SPLINE
SPL {X  -133.336, Y  +773.792, Z    +0.000, E1   -47.991, E3 +231264.760}
SPL {X  -153.017, Y  +738.949, Z    +0.000, E1   -37.928, E3 +231278.164}
SPL {X  -160.146, Y  +717.846, Z    +0.000, E1   -27.412, E3 +231265.710}
SPL {X  -163.639, Y  +701.236, Z    +0.000, E1   -18.901, E3 +231271.851}
SPL {X  -165.058, Y  +689.494, Z    +0.000, E1   -11.557, E3 +231270.668}
SPL {X  -165.574, Y  +680.514, Z    +0.000, E1    -5.500, E3 +231269.912}
SPL {X  -165.650, Y  +674.881, Z    +0.000, E1    -1.215, E3 +231269.515}
SPL {X  -165.650, Y  +672.727, Z    +0.000, E1    +0.658, E3 +231268.394}
SPL {X  -165.650, Y  +669.258, Z    +0.000, E1    +5.269, E3 +231267.747}
SPL {X  -165.650, Y  +665.011, Z    +0.000, E1   +11.627, E3 +231267.634}
SPL {X  -165.650, Y  +659.446, Z    +0.000, E1   +21.123, E3 +231266.498}
SPL {X  -165.650, Y  +651.038, Z    +0.000, E1   +34.281, E3 +231266.124}
SPL {X  -165.650, Y  +635.255, Z    +0.000, E1   +53.641, E3 +231264.312}
SPL {X  -165.650, Y  +581.672, Z    +0.000, E1   +69.744, E3 +231276.720}
SPL {X  -165.650, Y  +458.048, Z    +0.000, E1   +68.782, E3 +231357.453}
ENDSPLINE

SPLINE
SPL {X  -165.650, Y  +484.472, Z    +0.000, E1   +63.918, E3 +231371.703}
ENDSPLINE

SPLINE
SPL {X  -165.650, Y  +477.868, Z    +0.000, E1   +63.324, E3 +231382.881}
SPL {X  -165.650, Y  +463.578, Z    +0.000, E1   +63.625, E3 +231395.235}
SPL {X  -165.650, Y  +453.769, Z    +0.000, E1   +63.450, E3 +231406.493}
SPL {X  -165.650, Y  +444.234, Z    +0.000, E1   +63.262, E3 +231417.666}
SPL {X  -165.650, Y  +432.479, Z    +0.000, E1   +63.557, E3 +231427.486}
SPL {X  -165.650, Y  +422.068, Z    +0.000, E1   +63.630, E3 +231437.582}
SPL {X  -165.650, Y  +411.650, Z    +0.000, E1   +63.439, E3 +231449.600}
SPL {X  -165.650, Y  +399.089, Z    +0.000, E1   +63.334, E3 +231463.325}
ENDSPLINE

SPLINE
SPL {X  -165.650, Y  +410.094, Z    +0.000, E1   +60.049, E3 +231474.043}
ENDSPLINE

SPLINE
SPL {X  -165.650, Y  +398.700, Z    +0.000, E1   +60.415, E3 +231484.941}
SPL {X  -165.650, Y  +380.643, Z    +0.000, E1   +61.187, E3 +231500.302}
SPL {X  -165.125, Y  +365.326, Z    +0.000, E1   +61.696, E3 +231513.646}
SPL {X  -164.823, Y  +361.969, Z    +0.000, E1   +60.899, E3 +231522.881}
SPL {X  -163.414, Y  +351.372, Z    +0.000, E1   +61.284, E3 +231532.143}
SPL {X  -162.189, Y  +344.818, Z    +0.000, E1   +60.900, E3 +231541.996}
SPL {X  -160.769, Y  +338.584, Z    +0.000, E1   +60.413, E3 +231552.172}
SPL {X  -157.780, Y  +328.049, Z    +0.000, E1   +60.445, E3 +231563.839}
SPL {X  -155.286, Y  +320.826, Z    +0.000, E1   +59.686, E3 +231576.395}
SPL {X  -152.445, Y  +313.689, Z    +0.000, E1   +59.490, E3 +231585.460}
SPL {X  -149.851, Y  +307.898, Z    +0.000, E1   +58.978, E3 +231594.782}
SPL {X  -146.926, Y  +301.997, Z    +0.000, E1   +58.334, E3 +231604.744}
SPL {X  -143.997, Y  +296.618, Z    +0.000, E1   +58.069, E3 +231612.002}
SPL {X  -142.530, Y  +294.089, Z    +0.000, E1   +57.567, E3 +231617.185}
SPL {X  -134.010, Y  +281.128, Z    +0.000, E1   +60.923, E3 +231615.291}
SPL {X   -93.591, Y  +241.823, Z    +0.000, E1   +55.455, E3 +231707.829}
ENDSPLINE

SPLINE
SPL {X  -110.554, Y  +255.140, Z    +0.000, E1   +52.082, E3 +231834.785}
SPL {X  -137.038, Y  +285.439, Z    +0.000, E1   +46.261, E3 +231854.524}
SPL {X  -149.954, Y  +308.117, Z    +0.000, E1   +39.560, E3 +231860.872}
SPL {X  -160.070, Y  +335.868, Z    +0.000, E1   +27.320, E3 +231855.271}
SPL {X  -163.969, Y  +354.959, Z    +0.000, E1   +17.178, E3 +231855.785}
SPL {X  -165.261, Y  +367.153, Z    +0.000, E1    +9.611, E3 +231854.937}
SPL {X  -165.600, Y  +374.440, Z    +0.000, E1    +4.699, E3 +231854.199}
SPL {X  -165.650, Y  +379.657, Z    +0.000, E1    +0.819, E3 +231853.727}
SPL {X  -165.650, Y  +381.885, Z    +0.000, E1    -1.282, E3 +231852.971}
SPL {X  -165.650, Y  +386.855, Z    +0.000, E1    -7.700, E3 +231852.390}
SPL {X  -165.650, Y  +393.198, Z    +0.000, E1   -17.733, E3 +231851.366}
SPL {X  -165.650, Y  +399.991, Z    +0.000, E1   -27.922, E3 +231852.262}
SPL {X  -165.650, Y  +411.457, Z    +0.000, E1   -45.557, E3 +231848.010}
SPL {X  -165.650, Y  +427.627, Z    +0.000, E1   -58.747, E3 +231848.644}
SPL {X  -165.650, Y  +479.770, Z    +0.000, E1   -67.621, E3 +231869.258}
SPL {X  -165.650, Y  +594.725, Z    +0.000, E1   -69.155, E3 +231936.720}
ENDSPLINE

SPLINE
SPL {X  -165.650, Y  +562.482, Z    +0.000, E1   -62.785, E3 +231956.185}
ENDSPLINE

SPLINE
SPL {X  -165.650, Y  +572.898, Z    +0.000, E1   -62.409, E3 +231970.123}
SPL {X  -165.650, Y  +586.101, Z    +0.000, E1   -62.398, E3 +231984.194}
SPL {X  -165.650, Y  +596.110, Z    +0.000, E1   -62.302, E3 +231995.635}
SPL {X  -165.650, Y  +607.052, Z    +0.000, E1   -62.387, E3 +232006.702}
SPL {X  -165.650, Y  +615.372, Z    +0.000, E1   -62.260, E3 +232016.529}
SPL {X  -165.650, Y  +628.571, Z    +0.000, E1   -62.348, E3 +232030.250}
SPL {X  -165.650, Y  +640.498, Z    +0.000, E1   -62.343, E3 +232042.871}
SPL {X  -165.650, Y  +654.166, Z    +0.000, E1   -62.507, E3 +232056.522}
SPL {X  -165.650, Y  +665.926, Z    +0.000, E1   -62.171, E3 +232071.321}
SPL {X  -165.644, Y  +676.899, Z    +0.000, E1   -62.447, E3 +232081.088}
SPL {X  -165.241, Y  +687.133, Z    +0.000, E1   -62.230, E3 +232093.791}
SPL {X  -164.056, Y  +698.425, Z    +0.000, E1   -62.113, E3 +232106.607}
SPL {X  -162.891, Y  +705.608, Z    +0.000, E1   -61.899, E3 +232115.779}
SPL {X  -160.709, Y  +715.657, Z    +0.000, E1   -61.639, E3 +232128.531}
SPL {X  -157.706, Y  +726.183, Z    +0.000, E1   -61.153, E3 +232142.914}
SPL {X  -155.057, Y  +733.785, Z    +0.000, E1   -60.834, E3 +232152.904}
SPL {X  -152.882, Y  +739.274, Z    +0.000, E1   -60.485, E3 +232160.896}
SPL {X  -149.755, Y  +746.304, Z    +0.000, E1   -59.867, E3 +232172.017}
SPL {X  -146.068, Y  +753.629, Z    +0.000, E1   -59.384, E3 +232182.377}
SPL {X  -143.119, Y  +758.908, Z    +0.000, E1   -58.828, E3 +232190.751}
SPL {X  -141.017, Y  +762.414, Z    +0.000, E1   -58.435, E3 +232196.272}
SPL {X  -134.606, Y  +772.046, Z    +0.000, E1   -61.105, E3 +232193.918}
SPL {X  -127.075, Y  +781.763, Z    +0.000, E1   -62.555, E3 +232196.233}
SPL {X   -95.057, Y  +811.161, Z    +0.000, E1   -56.196, E3 +232276.286}
SPL {X   -88.361, Y  +815.615, Z    +0.000, E1   -54.176, E3 +232322.203}
ENDSPLINE

SPLINE
SPL {X  -120.253, Y  +789.426, Z    +0.000, E1   -51.165, E3 +232429.981}
SPL {X  -143.101, Y  +758.939, Z    +0.000, E1   -44.365, E3 +232444.089}
SPL {X  -158.740, Y  +722.846, Z    +0.000, E1   -30.140, E3 +232442.127}
SPL {X  -163.639, Y  +701.236, Z    +0.000, E1   -18.901, E3 +232444.265}
SPL {X  -165.058, Y  +689.494, Z    +0.000, E1   -11.557, E3 +232443.082}
SPL {X  -165.574, Y  +680.514, Z    +0.000, E1    -5.500, E3 +232442.326}
SPL {X  -165.650, Y  +673.883, Z    +0.000, E1    -0.454, E3 +232441.337}
SPL {X  -165.650, Y  +672.004, Z    +0.000, E1    +1.620, E3 +232440.543}
SPL {X  -165.650, Y  +669.258, Z    +0.000, E1    +5.269, E3 +232440.161}
SPL {X  -165.650, Y  +665.011, Z    +0.000, E1   +11.627, E3 +232440.048}
SPL {X  -165.650, Y  +659.446, Z    +0.000, E1   +21.123, E3 +232438.912}
SPL {X  -165.650, Y  +651.038, Z    +0.000, E1   +34.281, E3 +232438.538}
SPL {X  -165.650, Y  +635.255, Z    +0.000, E1   +53.641, E3 +232436.726}
SPL {X  -165.650, Y  +581.672, Z    +0.000, E1   +69.744, E3 +232449.134}
SPL {X  -165.650, Y  +458.048, Z    +0.000, E1   +68.782, E3 +232529.866}
ENDSPLINE

SPLINE
SPL {X  -165.650, Y  +484.472, Z    +0.000, E1   +63.918, E3 +232544.117}
ENDSPLINE

SPLINE
SPL {X  -165.650, Y  +477.868, Z    +0.000, E1   +63.324, E3 +232555.295}
SPL {X  -165.650, Y  +463.578, Z    +0.000, E1   +63.625, E3 +232567.649}
SPL {X  -165.650, Y  +453.769, Z    +0.000, E1   +63.450, E3 +232578.907}
SPL {X  -165.650, Y  +444.234, Z    +0.000, E1   +63.262, E3 +232590.080}
SPL {X  -165.650, Y  +432.479, Z    +0.000, E1   +63.557, E3 +232599.900}
SPL {X  -165.650, Y  +422.068, Z    +0.000, E1   +63.630, E3 +232609.995}
SPL {X  -165.650, Y  +411.650, Z    +0.000, E1   +63.439, E3 +232622.014}
SPL {X  -165.650, Y  +399.089, Z    +0.000, E1   +63.334, E3 +232635.739}
ENDSPLINE

SPLINE
SPL {X  -165.650, Y  +410.094, Z    +0.000, E1   +60.049, E3 +232646.456}
ENDSPLINE

SPLINE
SPL {X  -165.650, Y  +398.700, Z    +0.000, E1   +60.415, E3 +232657.354}
SPL {X  -165.650, Y  +380.643, Z    +0.000, E1   +61.187, E3 +232672.716}
SPL {X  -165.125, Y  +365.326, Z    +0.000, E1   +61.696, E3 +232686.060}
SPL {X  -164.823, Y  +361.969, Z    +0.000, E1   +60.899, E3 +232695.294}
SPL {X  -163.414, Y  +351.372, Z    +0.000, E1   +61.284, E3 +232704.557}
SPL {X  -162.189, Y  +344.818, Z    +0.000, E1   +60.900, E3 +232714.410}
SPL {X  -160.769, Y  +338.584, Z    +0.000, E1   +60.413, E3 +232724.586}
SPL {X  -157.780, Y  +328.049, Z    +0.000, E1   +60.445, E3 +232736.253}
SPL {X  -155.286, Y  +320.826, Z    +0.000, E1   +59.686, E3 +232748.809}
SPL {X  -152.445, Y  +313.689, Z    +0.000, E1   +59.490, E3 +232757.874}
SPL {X  -150.678, Y  +309.680, Z    +0.000, E1   +58.971, E3 +232765.186}
SPL {X  -148.010, Y  +304.117, Z    +0.000, E1   +58.696, E3 +232772.933}
SPL {X  -144.822, Y  +298.086, Z    +0.000, E1   +58.093, E3 +232782.715}
SPL {X  -142.530, Y  +294.089, Z    +0.000, E1   +57.567, E3 +232789.599}
SPL {X  -136.453, Y  +284.583, Z    +0.000, E1   +60.257, E3 +232787.410}
SPL {X  -128.205, Y  +273.602, Z    +0.000, E1   +62.388, E3 +232788.113}
SPL {X   -93.591, Y  +241.823, Z    +0.000, E1   +55.455, E3 +232880.243}
ENDSPLINE

SPLINE
SPL {X  -110.554, Y  +255.140, Z    +0.000, E1   +52.082, E3 +233007.199}
SPL {X  -137.038, Y  +285.439, Z    +0.000, E1   +46.261, E3 +233026.938}
SPL {X  -149.954, Y  +308.117, Z    +0.000, E1   +39.560, E3 +233033.286}
SPL {X  -160.070, Y  +335.868, Z    +0.000, E1   +27.320, E3 +233027.685}
SPL {X  -163.969, Y  +354.959, Z    +0.000, E1   +17.178, E3 +233028.199}
SPL {X  -165.261, Y  +367.153, Z    +0.000, E1    +9.611, E3 +233027.351}
SPL {X  -165.600, Y  +374.440, Z    +0.000, E1    +4.699, E3 +233026.612}
SPL {X  -165.650, Y  +379.657, Z    +0.000, E1    +0.819, E3 +233026.141}
SPL {X  -165.650, Y  +381.885, Z    +0.000, E1    -1.282, E3 +233025.385}
SPL {X  -165.650, Y  +386.855, Z    +0.000, E1    -7.700, E3 +233024.804}
SPL {X  -165.650, Y  +393.198, Z    +0.000, E1   -17.733, E3 +233023.780}
SPL {X  -165.650, Y  +399.991, Z    +0.000, E1   -27.922, E3 +233024.676}
SPL {X  -165.650, Y  +411.457, Z    +0.000, E1   -45.557, E3 +233020.424}
SPL {X  -165.650, Y  +427.627, Z    +0.000, E1   -58.747, E3 +233021.058}
SPL {X  -165.650, Y  +479.770, Z    +0.000, E1   -67.621, E3 +233041.672}
SPL {X  -165.650, Y  +594.725, Z    +0.000, E1   -69.155, E3 +233109.134}
ENDSPLINE

SPLINE
SPL {X  -165.650, Y  +565.175, Z    +0.000, E1   -62.653, E3 +233132.624}
ENDSPLINE

SPLINE
SPL {X  -165.650, Y  +576.067, Z    +0.000, E1   -62.373, E3 +233146.025}
SPL {X  -165.650, Y  +586.101, Z    +0.000, E1   -62.398, E3 +233156.608}
SPL {X  -165.650, Y  +596.110, Z    +0.000, E1   -62.302, E3 +233168.048}
SPL {X  -165.650, Y  +607.052, Z    +0.000, E1   -62.387, E3 +233179.116}
SPL {X  -165.650, Y  +618.920, Z    +0.000, E1   -62.340, E3 +233192.306}
SPL {X  -165.650, Y  +635.445, Z    +0.000, E1   -62.341, E3 +233210.106}
SPL {X  -165.650, Y  +654.166, Z    +0.000, E1   -62.507, E3 +233228.936}
SPL {X  -165.650, Y  +665.926, Z    +0.000, E1   -62.171, E3 +233243.734}
SPL {X  -165.644, Y  +676.899, Z    +0.000, E1   -62.447, E3 +233253.502}
SPL {X  -165.241, Y  +687.133, Z    +0.000, E1   -62.230, E3 +233266.204}
SPL {X  -164.056, Y  +698.425, Z    +0.000, E1   -62.113, E3 +233279.021}
SPL {X  -162.891, Y  +705.608, Z    +0.000, E1   -61.899, E3 +233288.193}
SPL {X  -161.308, Y  +713.180, Z    +0.000, E1   -61.813, E3 +233296.887}
SPL {X  -159.339, Y  +720.787, Z    +0.000, E1   -61.452, E3 +233307.582}
SPL {X  -156.103, Y  +730.922, Z    +0.000, E1   -60.875, E3 +233322.128}
SPL {X  -152.882, Y  +739.274, Z    +0.000, E1   -60.485, E3 +233333.310}
SPL {X  -150.387, Y  +744.953, Z    +0.000, E1   -60.023, E3 +233341.985}
SPL {X  -147.728, Y  +750.443, Z    +0.000, E1   -59.568, E3 +233350.369}
SPL {X  -143.895, Y  +757.561, Z    +0.000, E1   -58.980, E3 +233361.105}
SPL {X  -141.017, Y  +762.414, Z    +0.000, E1   -58.435, E3 +233368.685}
SPL {X  -132.386, Y  +775.068, Z    +0.000, E1   -61.559, E3 +233367.071}
SPL {X   -89.692, Y  +814.767, Z    +0.000, E1   -54.641, E3 +233481.120}
ENDSPLINE

SPLINE
SPL {X  -133.336, Y  +773.792, Z    +0.000, E1   -47.991, E3 +233609.587}
SPL {X  -153.017, Y  +738.949, Z    +0.000, E1   -37.928, E3 +233622.991}
SPL {X  -160.146, Y  +717.846, Z    +0.000, E1   -27.412, E3 +233610.537}
SPL {X  -163.639, Y  +701.236, Z    +0.000, E1   -18.901, E3 +233616.679}
SPL {X  -165.058, Y  +689.494, Z    +0.000, E1   -11.557, E3 +233615.496}
SPL {X  -165.574, Y  +680.514, Z    +0.000, E1    -5.500, E3 +233614.739}
SPL {X  -165.650, Y  +674.881, Z    +0.000, E1    -1.215, E3 +233614.342}
SPL {X  -165.650, Y  +673.425, Z    +0.000, E1    +0.051, E3 +233613.478}
SPL {X  -165.650, Y  +672.004, Z    +0.000, E1    +1.620, E3 +233612.956}
SPL {X  -165.650, Y  +669.258, Z    +0.000, E1    +5.269, E3 +233612.575}
SPL {X  -165.650, Y  +665.011, Z    +0.000, E1   +11.627, E3 +233612.462}
SPL {X  -165.650, Y  +659.446, Z    +0.000, E1   +21.123, E3 +233611.326}
SPL {X  -165.650, Y  +654.020, Z    +0.000, E1   +29.754, E3 +233611.481}
SPL {X  -165.650, Y  +644.843, Z    +0.000, E1   +43.427, E3 +233609.807}
SPL {X  -165.650, Y  +632.102, Z    +0.000, E1   +56.225, E3 +233609.155}
SPL {X  -165.650, Y  +581.672, Z    +0.000, E1   +69.744, E3 +233621.547}
SPL {X  -165.650, Y  +458.048, Z    +0.000, E1   +68.782, E3 +233702.280}
ENDSPLINE

SPLINE
SPL {X  -165.650, Y  +484.472, Z    +0.000, E1   +63.918, E3 +233716.531}
ENDSPLINE

SPLINE
SPL {X  -165.650, Y  +477.868, Z    +0.000, E1   +63.324, E3 +233727.708}
SPL {X  -165.650, Y  +463.578, Z    +0.000, E1   +63.625, E3 +233740.062}
SPL {X  -165.650, Y  +453.769, Z    +0.000, E1   +63.450, E3 +233751.321}
SPL {X  -165.650, Y  +444.234, Z    +0.000, E1   +63.262, E3 +233762.494}
SPL {X  -165.650, Y  +432.479, Z    +0.000, E1   +63.557, E3 +233772.314}
SPL {X  -165.650, Y  +422.068, Z    +0.000, E1   +63.630, E3 +233782.409}
SPL {X  -165.650, Y  +409.231, Z    +0.000, E1   +63.364, E3 +233797.658}
SPL {X  -165.650, Y  +395.008, Z    +0.000, E1   +63.445, E3 +233811.421}
ENDSPLINE

SPLINE
SPL {X  -165.650, Y  +410.094, Z    +0.000, E1   +60.049, E3 +233818.870}
ENDSPLINE

SPLINE
SPL {X  -165.650, Y  +398.700, Z    +0.000, E1   +60.415, E3 +233829.768}
SPL {X  -165.650, Y  +382.616, Z    +0.000, E1   +61.427, E3 +233840.987}
SPL {X  -165.650, Y  +379.013, Z    +0.000, E1   +60.888, E3 +233848.809}
SPL {X  -165.125, Y  +365.326, Z    +0.000, E1   +61.696, E3 +233858.473}
SPL {X  -164.823, Y  +361.969, Z    +0.000, E1   +60.899, E3 +233867.708}
SPL {X  -163.414, Y  +351.372, Z    +0.000, E1   +61.284, E3 +233876.971}
SPL {X  -162.189, Y  +344.818, Z    +0.000, E1   +60.900, E3 +233886.824}
SPL {X  -160.769, Y  +338.584, Z    +0.000, E1   +60.413, E3 +233897.000}
SPL {X  -157.780, Y  +328.049, Z    +0.000, E1   +60.445, E3 +233908.667}
SPL {X  -155.286, Y  +320.826, Z    +0.000, E1   +59.686, E3 +233921.222}
SPL {X  -152.445, Y  +313.689, Z    +0.000, E1   +59.490, E3 +233930.288}
SPL {X  -149.851, Y  +307.898, Z    +0.000, E1   +58.978, E3 +233939.610}
SPL {X  -146.926, Y  +301.997, Z    +0.000, E1   +58.334, E3 +233949.571}
SPL {X  -143.281, Y  +295.370, Z    +0.000, E1   +57.860, E3 +233959.340}
SPL {X  -136.453, Y  +284.583, Z    +0.000, E1   +60.257, E3 +233959.824}
SPL {X  -128.205, Y  +273.602, Z    +0.000, E1   +62.388, E3 +233960.527}
SPL {X   -93.591, Y  +241.823, Z    +0.000, E1   +55.455, E3 +234052.656}
ENDSPLINE

SPLINE
SPL {X  -110.554, Y  +255.140, Z    +0.000, E1   +52.082, E3 +234179.612}
SPL {X  -137.038, Y  +285.439, Z    +0.000, E1   +46.261, E3 +234199.352}
SPL {X  -149.954, Y  +308.117, Z    +0.000, E1   +39.560, E3 +234205.700}
SPL {X  -160.070, Y  +335.868, Z    +0.000, E1   +27.320, E3 +234200.098}
SPL {X  -163.969, Y  +354.959, Z    +0.000, E1   +17.178, E3 +234200.613}
SPL {X  -165.261, Y  +367.153, Z    +0.000, E1    +9.611, E3 +234199.765}
SPL {X  -165.600, Y  +374.440, Z    +0.000, E1    +4.699, E3 +234199.026}
SPL {X  -165.650, Y  +379.657, Z    +0.000, E1    +0.819, E3 +234198.555}
SPL {X  -165.650, Y  +381.885, Z    +0.000, E1    -1.282, E3 +234197.799}
SPL {X  -165.650, Y  +385.555, Z    +0.000, E1    -6.051, E3 +234196.944}
SPL {X  -165.650, Y  +388.884, Z    +0.000, E1   -10.835, E3 +234197.644}
SPL {X  -165.650, Y  +393.198, Z    +0.000, E1   -17.733, E3 +234196.194}
SPL {X  -165.650, Y  +399.991, Z    +0.000, E1   -27.922, E3 +234197.090}
SPL {X  -165.650, Y  +409.148, Z    +0.000, E1   -43.235, E3 +234192.476}
SPL {X  -165.650, Y  +420.563, Z    +0.000, E1   -54.059, E3 +234193.034}
SPL {X  -165.650, Y  +436.566, Z    +0.000, E1   -62.888, E3 +234194.747}
SPL {X  -165.650, Y  +479.770, Z    +0.000, E1   -67.621, E3 +234214.085}
SPL {X  -165.650, Y  +594.725, Z    +0.000, E1   -69.155, E3 +234281.547}
ENDSPLINE

SPLINE
SPL {X  -165.650, Y  +565.175, Z    +0.000, E1   -62.653, E3 +234305.038}
ENDSPLINE

SPLINE
SPL {X  -165.650, Y  +576.067, Z    +0.000, E1   -62.373, E3 +234318.439}
SPL {X  -165.650, Y  +586.101, Z    +0.000, E1   -62.398, E3 +234329.021}
SPL {X  -165.650, Y  +596.110, Z    +0.000, E1   -62.302, E3 +234340.462}
SPL {X  -165.650, Y  +607.052, Z    +0.000, E1   -62.387, E3 +234351.529}
SPL {X  -165.650, Y  +618.920, Z    +0.000, E1   -62.340, E3 +234364.720}
SPL {X  -165.650, Y  +635.445, Z    +0.000, E1   -62.341, E3 +234382.520}
SPL {X  -165.650, Y  +654.166, Z    +0.000, E1   -62.507, E3 +234401.350}
SPL {X  -165.650, Y  +665.926, Z    +0.000, E1   -62.171, E3 +234416.148}
SPL {X  -165.600, Y  +679.566, Z    +0.000, E1   -62.408, E3 +234429.186}
SPL {X  -165.066, Y  +689.394, Z    +0.000, E1   -62.143, E3 +234441.515}
SPL {X  -164.056, Y  +698.425, Z    +0.000, E1   -62.113, E3 +234451.435}
SPL {X  -162.891, Y  +705.608, Z    +0.000, E1   -61.899, E3 +234460.607}
SPL {X  -161.308, Y  +713.180, Z    +0.000, E1   -61.813, E3 +234469.300}
SPL {X  -159.339, Y  +720.787, Z    +0.000, E1   -61.452, E3 +234479.995}
SPL {X  -156.103, Y  +730.922, Z    +0.000, E1   -60.875, E3 +234494.542}
SPL {X  -152.882, Y  +739.274, Z    +0.000, E1   -60.485, E3 +234505.724}
SPL {X  -150.387, Y  +744.953, Z    +0.000, E1   -60.023, E3 +234514.399}
SPL {X  -147.728, Y  +750.443, Z    +0.000, E1   -59.568, E3 +234522.783}
SPL {X  -143.895, Y  +757.561, Z    +0.000, E1   -58.980, E3 +234533.519}
SPL {X  -141.017, Y  +762.414, Z    +0.000, E1   -58.435, E3 +234541.099}
SPL {X  -132.386, Y  +775.068, Z    +0.000, E1   -61.559, E3 +234539.485}
SPL {X   -89.692, Y  +814.767, Z    +0.000, E1   -54.641, E3 +234653.534}
ENDSPLINE

SPLINE
SPL {X  -133.336, Y  +773.792, Z    +0.000, E1   -47.991, E3 +234782.001}
SPL {X  -153.017, Y  +738.949, Z    +0.000, E1   -37.928, E3 +234795.405}
SPL {X  -160.146, Y  +717.846, Z    +0.000, E1   -27.412, E3 +234782.951}
SPL {X  -163.639, Y  +701.236, Z    +0.000, E1   -18.901, E3 +234789.093}
SPL {X  -165.058, Y  +689.494, Z    +0.000, E1   -11.557, E3 +234787.910}
SPL {X  -165.574, Y  +680.514, Z    +0.000, E1    -5.500, E3 +234787.153}
SPL {X  -165.650, Y  +673.883, Z    +0.000, E1    -0.454, E3 +234786.164}
SPL {X  -165.650, Y  +672.004, Z    +0.000, E1    +1.620, E3 +234785.370}
SPL {X  -165.650, Y  +669.258, Z    +0.000, E1    +5.269, E3 +234784.988}
SPL {X  -165.650, Y  +665.011, Z    +0.000, E1   +11.627, E3 +234784.876}
SPL {X  -165.650, Y  +659.446, Z    +0.000, E1   +21.123, E3 +234783.740}
SPL {X  -165.650, Y  +654.020, Z    +0.000, E1   +29.754, E3 +234783.894}
SPL {X  -165.650, Y  +644.843, Z    +0.000, E1   +43.427, E3 +234782.220}
SPL {X  -165.650, Y  +632.102, Z    +0.000, E1   +56.225, E3 +234781.569}
SPL {X  -165.650, Y  +581.672, Z    +0.000, E1   +69.744, E3 +234793.961}
SPL {X  -165.650, Y  +458.048, Z    +0.000, E1   +68.782, E3 +234874.694}
ENDSPLINE

SPLINE
SPL {X  -165.650, Y  +484.472, Z    +0.000, E1   +63.918, E3 +234888.945}
ENDSPLINE

SPLINE
SPL {X  -165.650, Y  +477.868, Z    +0.000, E1   +63.324, E3 +234900.122}
SPL {X  -165.650, Y  +463.578, Z    +0.000, E1   +63.625, E3 +234912.476}
SPL {X  -165.650, Y  +453.769, Z    +0.000, E1   +63.450, E3 +234923.735}
SPL {X  -165.650, Y  +444.234, Z    +0.000, E1   +63.262, E3 +234934.908}
SPL {X  -165.650, Y  +432.479, Z    +0.000, E1   +63.557, E3 +234944.728}
SPL {X  -165.650, Y  +422.068, Z    +0.000, E1   +63.630, E3 +234954.823}
SPL {X  -165.650, Y  +409.231, Z    +0.000, E1   +63.364, E3 +234970.071}
SPL {X  -165.650, Y  +395.008, Z    +0.000, E1   +63.445, E3 +234983.835}
ENDSPLINE

SPLINE
SPL {X  -165.650, Y  +410.094, Z    +0.000, E1   +60.049, E3 +234991.284}
ENDSPLINE

SPLINE
SPL {X  -165.650, Y  +398.700, Z    +0.000, E1   +60.415, E3 +235002.182}
SPL {X  -165.650, Y  +382.616, Z    +0.000, E1   +61.427, E3 +235013.400}
SPL {X  -165.650, Y  +379.013, Z    +0.000, E1   +60.888, E3 +235021.223}
SPL {X  -165.125, Y  +365.326, Z    +0.000, E1   +61.696, E3 +235030.887}
SPL {X  -164.823, Y  +361.969, Z    +0.000, E1   +60.899, E3 +235040.122}
SPL {X  -163.414, Y  +351.372, Z    +0.000, E1   +61.284, E3 +235049.385}
SPL {X  -162.189, Y  +344.818, Z    +0.000, E1   +60.900, E3 +235059.238}
SPL {X  -160.769, Y  +338.584, Z    +0.000, E1   +60.413, E3 +235069.414}
SPL {X  -157.780, Y  +328.049, Z    +0.000, E1   +60.445, E3 +235081.081}
SPL {X  -155.286, Y  +320.826, Z    +0.000, E1   +59.686, E3 +235093.636}
SPL {X  -152.445, Y  +313.689, Z    +0.000, E1   +59.490, E3 +235102.702}
SPL {X  -149.851, Y  +307.898, Z    +0.000, E1   +58.978, E3 +235112.024}
SPL {X  -146.926, Y  +301.997, Z    +0.000, E1   +58.334, E3 +235121.985}
SPL {X  -143.997, Y  +296.618, Z    +0.000, E1   +58.069, E3 +235129.243}
SPL {X  -142.530, Y  +294.089, Z    +0.000, E1   +57.567, E3 +235134.426}
SPL {X  -134.010, Y  +281.128, Z    +0.000, E1   +60.923, E3 +235132.532}
SPL {X   -93.591, Y  +241.823, Z    +0.000, E1   +55.455, E3 +235225.070}
ENDSPLINE

SPLINE
SPL {X  -110.554, Y  +255.140, Z    +0.000, E1   +52.082, E3 +235352.026}
SPL {X  -144.988, Y  +298.385, Z    +0.000, E1   +42.755, E3 +235375.845}
SPL {X  -160.070, Y  +335.868, Z    +0.000, E1   +27.320, E3 +235372.512}
SPL {X  -163.969, Y  +354.959, Z    +0.000, E1   +17.178, E3 +235373.026}
SPL {X  -165.261, Y  +367.153, Z    +0.000, E1    +9.611, E3 +235372.179}
SPL {X  -165.600, Y  +374.440, Z    +0.000, E1    +4.699, E3 +235371.440}
SPL {X  -165.650, Y  +379.657, Z    +0.000, E1    +0.819, E3 +235370.968}
SPL {X  -165.650, Y  +381.885, Z    +0.000, E1    -1.282, E3 +235370.213}
SPL {X  -165.650, Y  +386.855, Z    +0.000, E1    -7.700, E3 +235369.632}
SPL {X  -165.650, Y  +393.198, Z    +0.000, E1   -17.733, E3 +235368.608}
SPL {X  -165.650, Y  +399.991, Z    +0.000, E1   -27.922, E3 +235369.503}
SPL {X  -165.650, Y  +409.148, Z    +0.000, E1   -43.235, E3 +235364.890}
SPL {X  -165.650, Y  +420.563, Z    +0.000, E1   -54.059, E3 +235365.447}
SPL {X  -165.650, Y  +436.566, Z    +0.000, E1   -62.888, E3 +235367.160}
SPL {X  -165.650, Y  +479.770, Z    +0.000, E1   -67.621, E3 +235386.499}
SPL {X  -165.650, Y  +594.725, Z    +0.000, E1   -69.155, E3 +235453.961}
ENDSPLINE

SPLINE
SPL {X  -165.650, Y  +565.175, Z    +0.000, E1   -62.653, E3 +235477.452}
ENDSPLINE

SPLINE
SPL {X  -165.650, Y  +576.067, Z    +0.000, E1   -62.373, E3 +235490.853}
SPL {X  -165.650, Y  +586.101, Z    +0.000, E1   -62.398, E3 +235501.435}
SPL {X  -165.650, Y  +596.110, Z    +0.000, E1   -62.302, E3 +235512.876}
SPL {X  -165.650, Y  +607.052, Z    +0.000, E1   -62.387, E3 +235523.943}
SPL {X  -165.650, Y  +618.920, Z    +0.000, E1   -62.340, E3 +235537.133}
SPL {X  -165.650, Y  +635.445, Z    +0.000, E1   -62.341, E3 +235554.934}
SPL {X  -165.650, Y  +654.166, Z    +0.000, E1   -62.507, E3 +235573.764}
SPL {X  -165.650, Y  +665.926, Z    +0.000, E1   -62.171, E3 +235588.562}
SPL {X  -165.644, Y  +676.899, Z    +0.000, E1   -62.447, E3 +235598.329}
SPL {X  -165.241, Y  +687.133, Z    +0.000, E1   -62.230, E3 +235611.032}
SPL {X  -164.056, Y  +698.425, Z    +0.000, E1   -62.113, E3 +235623.849}
SPL {X  -162.891, Y  +705.608, Z    +0.000, E1   -61.899, E3 +235633.020}
SPL {X  -160.709, Y  +715.657, Z    +0.000, E1   -61.639, E3 +235645.772}
SPL {X  -157.706, Y  +726.183, Z    +0.000, E1   -61.153, E3 +235660.155}
SPL {X  -155.057, Y  +733.785, Z    +0.000, E1   -60.834, E3 +235670.145}
SPL {X  -152.882, Y  +739.274, Z    +0.000, E1   -60.485, E3 +235678.137}
SPL {X  -150.387, Y  +744.953, Z    +0.000, E1   -60.023, E3 +235686.812}
SPL {X  -147.728, Y  +750.443, Z    +0.000, E1   -59.568, E3 +235695.196}
SPL {X  -143.895, Y  +757.561, Z    +0.000, E1   -58.980, E3 +235705.933}
SPL {X  -141.017, Y  +762.414, Z    +0.000, E1   -58.435, E3 +235713.513}
SPL {X  -134.606, Y  +772.046, Z    +0.000, E1   -61.105, E3 +235711.160}
SPL {X  -127.075, Y  +781.763, Z    +0.000, E1   -62.555, E3 +235713.474}
SPL {X   -89.692, Y  +814.767, Z    +0.000, E1   -54.641, E3 +235825.948}
ENDSPLINE

SPLINE
SPL {X  -133.336, Y  +773.792, Z    +0.000, E1   -47.991, E3 +235954.415}
SPL {X  -153.017, Y  +738.949, Z    +0.000, E1   -37.928, E3 +235967.819}
SPL {X  -160.146, Y  +717.846, Z    +0.000, E1   -27.412, E3 +235955.365}
SPL {X  -163.639, Y  +701.236, Z    +0.000, E1   -18.901, E3 +235961.506}
SPL {X  -165.380, Y  +684.951, Z    +0.000, E1    -8.606, E3 +235959.764}
SPL {X  -165.650, Y  +675.640, Z    +0.000, E1    -1.874, E3 +235959.300}
SPL {X  -165.650, Y  +672.727, Z    +0.000, E1    +0.658, E3 +235958.049}
SPL {X  -165.650, Y  +669.258, Z    +0.000, E1    +5.269, E3 +235957.402}
SPL {X  -165.650, Y  +665.011, Z    +0.000, E1   +11.627, E3 +235957.289}
SPL {X  -165.650, Y  +659.446, Z    +0.000, E1   +21.123, E3 +235956.154}
SPL {X  -165.650, Y  +654.020, Z    +0.000, E1   +29.754, E3 +235956.308}
SPL {X  -165.650, Y  +644.843, Z    +0.000, E1   +43.427, E3 +235954.634}
SPL {X  -165.650, Y  +632.102, Z    +0.000, E1   +56.225, E3 +235953.983}
SPL {X  -165.650, Y  +581.672, Z    +0.000, E1   +69.744, E3 +235966.375}
SPL {X  -165.650, Y  +455.882, Z    +0.000, E1   +70.075, E3 +236038.640}
ENDSPLINE

SPLINE
SPL {X  -165.650, Y  +480.501, Z    +0.000, E1   +64.561, E3 +236060.609}
ENDSPLINE

SPLINE
SPL {X  -165.650, Y  +477.868, Z    +0.000, E1   +63.324, E3 +236072.536}
SPL {X  -165.650, Y  +463.578, Z    +0.000, E1   +63.625, E3 +236084.890}
SPL {X  -165.650, Y  +453.769, Z    +0.000, E1   +63.450, E3 +236096.149}
SPL {X  -165.650, Y  +444.234, Z    +0.000, E1   +63.262, E3 +236107.321}
SPL {X  -165.650, Y  +432.479, Z    +0.000, E1   +63.557, E3 +236117.141}
SPL {X  -165.650, Y  +422.068, Z    +0.000, E1   +63.630, E3 +236127.237}
SPL {X  -165.650, Y  +409.231, Z    +0.000, E1   +63.364, E3 +236142.485}
SPL {X  -165.650, Y  +395.008, Z    +0.000, E1   +63.445, E3 +236156.249}
ENDSPLINE

SPLINE
SPL {X  -165.650, Y  +410.094, Z    +0.000, E1   +60.049, E3 +236163.698}
ENDSPLINE

SPLINE
SPL {X  -165.650, Y  +398.700, Z    +0.000, E1   +60.415, E3 +236174.596}
SPL {X  -165.650, Y  +380.643, Z    +0.000, E1   +61.187, E3 +236189.957}
SPL {X  -165.125, Y  +365.326, Z    +0.000, E1   +61.696, E3 +236203.301}
SPL {X  -164.823, Y  +361.969, Z    +0.000, E1   +60.899, E3 +236212.536}
SPL {X  -163.414, Y  +351.372, Z    +0.000, E1   +61.284, E3 +236221.798}
SPL {X  -162.189, Y  +344.818, Z    +0.000, E1   +60.900, E3 +236231.652}
SPL {X  -160.769, Y  +338.584, Z    +0.000, E1   +60.413, E3 +236241.828}
SPL {X  -157.780, Y  +328.049, Z    +0.000, E1   +60.445, E3 +236253.494}
SPL {X  -155.286, Y  +320.826, Z    +0.000, E1   +59.686, E3 +236266.050}
SPL {X  -152.445, Y  +313.689, Z    +0.000, E1   +59.490, E3 +236275.115}
SPL {X  -149.851, Y  +307.898, Z    +0.000, E1   +58.978, E3 +236284.438}
SPL {X  -146.926, Y  +301.997, Z    +0.000, E1   +58.334, E3 +236294.399}
SPL {X  -143.281, Y  +295.370, Z    +0.000, E1   +57.860, E3 +236304.167}
SPL {X  -134.010, Y  +281.128, Z    +0.000, E1   +60.923, E3 +236304.946}
SPL {X   -93.591, Y  +241.823, Z    +0.000, E1   +55.455, E3 +236397.484}
ENDSPLINE

SPLINE
SPL {X  -110.554, Y  +255.140, Z    +0.000, E1   +52.082, E3 +236524.440}
SPL {X  -137.038, Y  +285.439, Z    +0.000, E1   +46.261, E3 +236544.180}
SPL {X  -149.954, Y  +308.117, Z    +0.000, E1   +39.560, E3 +236550.527}
SPL {X  -160.070, Y  +335.868, Z    +0.000, E1   +27.320, E3 +236544.926}
SPL {X  -163.969, Y  +354.959, Z    +0.000, E1   +17.178, E3 +236545.440}
SPL {X  -165.261, Y  +367.153, Z    +0.000, E1    +9.611, E3 +236544.593}
SPL {X  -165.600, Y  +374.440, Z    +0.000, E1    +4.699, E3 +236543.854}
SPL {X  -165.650, Y  +379.657, Z    +0.000, E1    +0.819, E3 +236543.382}
SPL {X  -165.650, Y  +381.885, Z    +0.000, E1    -1.282, E3 +236542.626}
SPL {X  -165.650, Y  +386.855, Z    +0.000, E1    -7.700, E3 +236542.045}
SPL {X  -165.650, Y  +393.198, Z    +0.000, E1   -17.733, E3 +236541.021}
SPL {X  -165.650, Y  +399.991, Z    +0.000, E1   -27.922, E3 +236541.917}
SPL {X  -165.650, Y  +409.148, Z    +0.000, E1   -43.235, E3 +236537.303}
SPL {X  -165.650, Y  +420.563, Z    +0.000, E1   -54.059, E3 +236537.861}
SPL {X  -165.650, Y  +436.566, Z    +0.000, E1   -62.888, E3 +236539.574}
SPL {X  -165.650, Y  +479.770, Z    +0.000, E1   -67.621, E3 +236558.913}
SPL {X  -165.650, Y  +594.725, Z    +0.000, E1   -69.155, E3 +236626.375}
ENDSPLINE

SPLINE
SPL {X  -165.650, Y  +565.175, Z    +0.000, E1   -62.653, E3 +236649.866}
ENDSPLINE

SPLINE
SPL {X  -165.650, Y  +576.067, Z    +0.000, E1   -62.373, E3 +236663.267}
SPL {X  -165.650, Y  +586.101, Z    +0.000, E1   -62.398, E3 +236673.849}
SPL {X  -165.650, Y  +596.110, Z    +0.000, E1   -62.302, E3 +236685.290}
SPL {X  -165.650, Y  +607.052, Z    +0.000, E1   -62.387, E3 +236696.357}
SPL {X  -165.650, Y  +618.920, Z    +0.000, E1   -62.340, E3 +236709.547}
SPL {X  -165.650, Y  +631.247, Z    +0.000, E1   -62.270, E3 +236723.164}
SPL {X  -165.650, Y  +645.288, Z    +0.000, E1   -62.475, E3 +236736.844}
SPL {X  -165.650, Y  +657.265, Z    +0.000, E1   -62.410, E3 +236749.962}
SPL {X  -165.650, Y  +665.926, Z    +0.000, E1   -62.171, E3 +236760.976}
SPL {X  -165.644, Y  +676.899, Z    +0.000, E1   -62.447, E3 +236770.743}
SPL {X  -165.241, Y  +687.133, Z    +0.000, E1   -62.230, E3 +236783.446}
SPL {X  -164.056, Y  +698.425, Z    +0.000, E1   -62.113, E3 +236796.263}
SPL {X  -162.891, Y  +705.608, Z    +0.000, E1   -61.899, E3 +236805.434}
SPL {X  -160.709, Y  +715.657, Z    +0.000, E1   -61.639, E3 +236818.186}
SPL {X  -157.706, Y  +726.183, Z    +0.000, E1   -61.153, E3 +236832.569}
SPL {X  -155.057, Y  +733.785, Z    +0.000, E1   -60.834, E3 +236842.559}
SPL {X  -152.882, Y  +739.274, Z    +0.000, E1   -60.485, E3 +236850.551}
SPL {X  -150.387, Y  +744.953, Z    +0.000, E1   -60.023, E3 +236859.226}
SPL {X  -146.839, Y  +752.170, Z    +0.000, E1   -59.458, E3 +236870.185}
SPL {X  -142.415, Y  +760.104, Z    +0.000, E1   -58.730, E3 +236882.244}
SPL {X  -132.386, Y  +775.068, Z    +0.000, E1   -61.559, E3 +236884.312}
SPL {X   -89.692, Y  +814.767, Z    +0.000, E1   -54.641, E3 +236998.362}
ENDSPLINE

SPLINE
SPL {X  -120.253, Y  +789.426, Z    +0.000, E1   -51.165, E3 +237119.636}
SPL {X  -143.101, Y  +758.939, Z    +0.000, E1   -44.365, E3 +237133.744}
SPL {X  -158.740, Y  +722.846, Z    +0.000, E1   -30.140, E3 +237131.782}
SPL {X  -163.639, Y  +701.236, Z    +0.000, E1   -18.901, E3 +237133.920}
SPL {X  -165.058, Y  +689.494, Z    +0.000, E1   -11.557, E3 +237132.737}
SPL {X  -165.574, Y  +680.514, Z    +0.000, E1    -5.500, E3 +237131.981}
SPL {X  -165.650, Y  +673.883, Z    +0.000, E1    -0.454, E3 +237130.992}
SPL {X  -165.650, Y  +672.004, Z    +0.000, E1    +1.620, E3 +237130.198}
SPL {X  -165.650, Y  +669.258, Z    +0.000, E1    +5.269, E3 +237129.816}
SPL {X  -165.650, Y  +665.011, Z    +0.000, E1   +11.627, E3 +237129.703}
SPL {X  -165.650, Y  +659.446, Z    +0.000, E1   +21.123, E3 +237128.567}
SPL {X  -165.650, Y  +654.020, Z    +0.000, E1   +29.754, E3 +237128.722}
SPL {X  -165.650, Y  +644.843, Z    +0.000, E1   +43.427, E3 +237127.048}
SPL {X  -165.650, Y  +632.102, Z    +0.000, E1   +56.225, E3 +237126.397}
SPL {X  -165.650, Y  +581.672, Z    +0.000, E1   +69.744, E3 +237138.789}
SPL {X  -165.650, Y  +458.048, Z    +0.000, E1   +68.782, E3 +237219.522}
ENDSPLINE

SPLINE
SPL {X  -165.650, Y  +484.472, Z    +0.000, E1   +63.918, E3 +237233.772}
ENDSPLINE

SPLINE
SPL {X  -165.650, Y  +477.868, Z    +0.000, E1   +63.324, E3 +237244.950}
SPL {X  -165.650, Y  +463.578, Z    +0.000, E1   +63.625, E3 +237257.304}
SPL {X  -165.650, Y  +453.769, Z    +0.000, E1   +63.450, E3 +237268.562}
SPL {X  -165.650, Y  +444.234, Z    +0.000, E1   +63.262, E3 +237279.735}
SPL {X  -165.650, Y  +432.479, Z    +0.000, E1   +63.557, E3 +237289.555}
SPL {X  -165.650, Y  +422.068, Z    +0.000, E1   +63.630, E3 +237299.650}
SPL {X  -165.650, Y  +411.650, Z    +0.000, E1   +63.439, E3 +237311.669}
SPL {X  -165.650, Y  +399.089, Z    +0.000, E1   +63.334, E3 +237325.394}
ENDSPLINE

SPLINE
SPL {X  -165.650, Y  +410.094, Z    +0.000, E1   +60.049, E3 +237336.112}
ENDSPLINE

SPLINE
SPL {X  -165.650, Y  +398.700, Z    +0.000, E1   +60.415, E3 +237347.010}
SPL {X  -165.650, Y  +380.643, Z    +0.000, E1   +61.187, E3 +237362.371}
SPL {X  -165.125, Y  +365.326, Z    +0.000, E1   +61.696, E3 +237375.715}
SPL {X  -164.823, Y  +361.969, Z    +0.000, E1   +60.899, E3 +237384.950}
SPL {X  -163.414, Y  +351.372, Z    +0.000, E1   +61.284, E3 +237394.212}
SPL {X  -162.189, Y  +344.818, Z    +0.000, E1   +60.900, E3 +237404.065}
SPL {X  -160.769, Y  +338.584, Z    +0.000, E1   +60.413, E3 +237414.241}
SPL {X  -157.780, Y  +328.049, Z    +0.000, E1   +60.445, E3 +237425.908}
SPL {X  -155.286, Y  +320.826, Z    +0.000, E1   +59.686, E3 +237438.464}
SPL {X  -152.445, Y  +313.689, Z    +0.000, E1   +59.490, E3 +237447.529}
SPL {X  -149.851, Y  +307.898, Z    +0.000, E1   +58.978, E3 +237456.851}
SPL {X  -146.926, Y  +301.997, Z    +0.000, E1   +58.334, E3 +237466.813}
SPL {X  -143.997, Y  +296.618, Z    +0.000, E1   +58.069, E3 +237474.071}
SPL {X  -142.530, Y  +294.089, Z    +0.000, E1   +57.567, E3 +237479.254}
SPL {X  -134.010, Y  +281.128, Z    +0.000, E1   +60.923, E3 +237477.360}
SPL {X   -93.591, Y  +241.823, Z    +0.000, E1   +55.455, E3 +237569.898}
ENDSPLINE

SPLINE
SPL {X  -110.554, Y  +255.140, Z    +0.000, E1   +52.082, E3 +237696.854}
SPL {X  -137.038, Y  +285.439, Z    +0.000, E1   +46.261, E3 +237716.593}
SPL {X  -149.954, Y  +308.117, Z    +0.000, E1   +39.560, E3 +237722.941}
SPL {X  -160.070, Y  +335.868, Z    +0.000, E1   +27.320, E3 +237717.340}
SPL {X  -163.969, Y  +354.959, Z    +0.000, E1   +17.178, E3 +237717.854}
SPL {X  -165.261, Y  +367.153, Z    +0.000, E1    +9.611, E3 +237717.006}
SPL {X  -165.600, Y  +374.440, Z    +0.000, E1    +4.699, E3 +237716.268}
SPL {X  -165.650, Y  +380.303, Z    +0.000, E1    +0.337, E3 +237715.478}
SPL {X  -165.650, Y  +382.684, Z    +0.000, E1    -2.314, E3 +237714.973}
SPL {X  -165.650, Y  +385.555, Z    +0.000, E1    -6.051, E3 +237714.186}
SPL {X  -165.650, Y  +388.884, Z    +0.000, E1   -10.835, E3 +237714.886}
SPL {X  -165.650, Y  +393.198, Z    +0.000, E1   -17.733, E3 +237713.435}
SPL {X  -165.650, Y  +399.991, Z    +0.000, E1   -27.922, E3 +237714.331}
SPL {X  -165.650, Y  +409.148, Z    +0.000, E1   -43.235, E3 +237709.717}
SPL {X  -165.650, Y  +420.563, Z    +0.000, E1   -54.059, E3 +237710.275}
SPL {X  -165.650, Y  +436.566, Z    +0.000, E1   -62.888, E3 +237711.988}
SPL {X  -165.650, Y  +479.770, Z    +0.000, E1   -67.621, E3 +237731.327}
SPL {X  -165.650, Y  +594.725, Z    +0.000, E1   -69.155, E3 +237798.789}
ENDSPLINE

SPLINE
SPL {X  -165.650, Y  +565.175, Z    +0.000, E1   -62.653, E3 +237822.279}
ENDSPLINE

SPLINE
SPL {X  -165.650, Y  +576.067, Z    +0.000, E1   -62.373, E3 +237835.681}
SPL {X  -165.650, Y  +586.101, Z    +0.000, E1   -62.398, E3 +237846.263}
SPL {X  -165.650, Y  +596.110, Z    +0.000, E1   -62.302, E3 +237857.704}
SPL {X  -165.650, Y  +607.052, Z    +0.000, E1   -62.387, E3 +237868.771}
SPL {X  -165.650, Y  +618.920, Z    +0.000, E1   -62.340, E3 +237881.961}
SPL {X  -165.650, Y  +631.247, Z    +0.000, E1   -62.270, E3 +237895.577}
SPL {X  -165.650, Y  +645.288, Z    +0.000, E1   -62.475, E3 +237909.258}
SPL {X  -165.650, Y  +657.265, Z    +0.000, E1   -62.410, E3 +237922.376}
SPL {X  -165.650, Y  +665.926, Z    +0.000, E1   -62.171, E3 +237933.390}
SPL {X  -165.600, Y  +679.566, Z    +0.000, E1   -62.408, E3 +237946.427}
SPL {X  -165.066, Y  +689.394, Z    +0.000, E1   -62.143, E3 +237958.756}
SPL {X  -164.056, Y  +698.425, Z    +0.000, E1   -62.113, E3 +237968.676}
SPL {X  -162.891, Y  +705.608, Z    +0.000, E1   -61.899, E3 +237977.848}
SPL {X  -160.709, Y  +715.657, Z    +0.000, E1   -61.639, E3 +237990.600}
SPL {X  -157.706, Y  +726.183, Z    +0.000, E1   -61.153, E3 +238004.983}
SPL {X  -155.057, Y  +733.785, Z    +0.000, E1   -60.834, E3 +238014.973}
SPL {X  -152.882, Y  +739.274, Z    +0.000, E1   -60.485, E3 +238022.965}
SPL {X  -150.387, Y  +744.953, Z    +0.000, E1   -60.023, E3 +238031.640}
SPL {X  -146.839, Y  +752.170, Z    +0.000, E1   -59.458, E3 +238042.599}
SPL {X  -142.415, Y  +760.104, Z    +0.000, E1   -58.730, E3 +238054.658}
SPL {X  -132.386, Y  +775.068, Z    +0.000, E1   -61.559, E3 +238056.726}
SPL {X   -89.692, Y  +814.767, Z    +0.000, E1   -54.641, E3 +238170.775}
ENDSPLINE

SPLINE
SPL {X  -133.336, Y  +773.792, Z    +0.000, E1   -47.991, E3 +238299.242}
SPL {X  -153.017, Y  +738.949, Z    +0.000, E1   -37.928, E3 +238312.646}
SPL {X  -160.146, Y  +717.846, Z    +0.000, E1   -27.412, E3 +238300.193}
SPL {X  -163.639, Y  +701.236, Z    +0.000, E1   -18.901, E3 +238306.334}
SPL {X  -165.380, Y  +684.951, Z    +0.000, E1    -8.606, E3 +238304.591}
SPL {X  -165.650, Y  +675.640, Z    +0.000, E1    -1.874, E3 +238304.127}
SPL {X  -165.650, Y  +672.727, Z    +0.000, E1    +0.658, E3 +238302.877}
SPL {X  -165.650, Y  +669.258, Z    +0.000, E1    +5.269, E3 +238302.230}
SPL {X  -165.650, Y  +665.011, Z    +0.000, E1   +11.627, E3 +238302.117}
SPL {X  -165.650, Y  +659.446, Z    +0.000, E1   +21.123, E3 +238300.981}
SPL {X  -165.650, Y  +654.020, Z    +0.000, E1   +29.754, E3 +238301.136}
SPL {X  -165.650, Y  +644.843, Z    +0.000, E1   +43.427, E3 +238299.462}
SPL {X  -165.650, Y  +632.102, Z    +0.000, E1   +56.225, E3 +238298.810}
SPL {X  -165.650, Y  +581.672, Z    +0.000, E1   +69.744, E3 +238311.203}
SPL {X  -165.650, Y  +458.048, Z    +0.000, E1   +68.782, E3 +238391.935}
ENDSPLINE

SPLINE
SPL {X  -165.650, Y  +484.472, Z    +0.000, E1   +63.918, E3 +238406.186}
ENDSPLINE

SPLINE
SPL {X  -165.650, Y  +477.868, Z    +0.000, E1   +63.324, E3 +238417.364}
SPL {X  -165.650, Y  +463.578, Z    +0.000, E1   +63.625, E3 +238429.718}
SPL {X  -165.650, Y  +453.769, Z    +0.000, E1   +63.450, E3 +238440.976}
SPL {X  -165.650, Y  +444.234, Z    +0.000, E1   +63.262, E3 +238452.149}
SPL {X  -165.650, Y  +432.479, Z    +0.000, E1   +63.557, E3 +238461.969}
SPL {X  -165.650, Y  +422.068, Z    +0.000, E1   +63.630, E3 +238472.064}
SPL {X  -165.650, Y  +411.650, Z    +0.000, E1   +63.439, E3 +238484.083}
SPL {X  -165.650, Y  +399.089, Z    +0.000, E1   +63.334, E3 +238497.808}
ENDSPLINE

SPLINE
SPL {X  -165.650, Y  +410.094, Z    +0.000, E1   +60.049, E3 +238508.525}
ENDSPLINE

SPLINE
SPL {X  -165.650, Y  +398.700, Z    +0.000, E1   +60.415, E3 +238519.423}
SPL {X  -165.650, Y  +382.616, Z    +0.000, E1   +61.427, E3 +238530.642}
SPL {X  -165.650, Y  +379.013, Z    +0.000, E1   +60.888, E3 +238538.464}
SPL {X  -165.125, Y  +365.326, Z    +0.000, E1   +61.696, E3 +238548.129}
SPL {X  -164.823, Y  +361.969, Z    +0.000, E1   +60.899, E3 +238557.363}
SPL {X  -163.414, Y  +351.372, Z    +0.000, E1   +61.284, E3 +238566.626}
SPL {X  -162.189, Y  +344.818, Z    +0.000, E1   +60.900, E3 +238576.479}
SPL {X  -160.769, Y  +338.584, Z    +0.000, E1   +60.413, E3 +238586.655}
SPL {X  -158.568, Y  +330.583, Z    +0.000, E1   +60.533, E3 +238594.795}
SPL {X  -157.003, Y  +325.679, Z    +0.000, E1   +60.284, E3 +238601.765}
SPL {X  -155.286, Y  +320.826, Z    +0.000, E1   +59.686, E3 +238610.878}
SPL {X  -152.445, Y  +313.689, Z    +0.000, E1   +59.490, E3 +238619.943}
SPL {X  -150.678, Y  +309.680, Z    +0.000, E1   +58.971, E3 +238627.255}
SPL {X  -148.010, Y  +304.117, Z    +0.000, E1   +58.696, E3 +238635.002}
SPL {X  -144.822, Y  +298.086, Z    +0.000, E1   +58.093, E3 +238644.784}
SPL {X  -142.530, Y  +294.089, Z    +0.000, E1   +57.567, E3 +238651.668}
SPL {X  -134.010, Y  +281.128, Z    +0.000, E1   +60.923, E3 +238649.773}
SPL {X   -93.591, Y  +241.823, Z    +0.000, E1   +55.455, E3 +238742.312}
ENDSPLINE

SPLINE
SPL {X  -110.554, Y  +255.140, Z    +0.000, E1   +52.082, E3 +238869.268}
SPL {X  -137.038, Y  +285.439, Z    +0.000, E1   +46.261, E3 +238889.007}
SPL {X  -149.954, Y  +308.117, Z    +0.000, E1   +39.560, E3 +238895.355}
SPL {X  -160.070, Y  +335.868, Z    +0.000, E1   +27.320, E3 +238889.754}
SPL {X  -163.969, Y  +354.959, Z    +0.000, E1   +17.178, E3 +238890.268}
SPL {X  -165.261, Y  +367.153, Z    +0.000, E1    +9.611, E3 +238889.420}
SPL {X  -165.600, Y  +374.440, Z    +0.000, E1    +4.699, E3 +238888.681}
SPL {X  -165.650, Y  +379.657, Z    +0.000, E1    +0.819, E3 +238888.210}
SPL {X  -165.650, Y  +381.885, Z    +0.000, E1    -1.282, E3 +238887.454}
SPL {X  -165.650, Y  +386.855, Z    +0.000, E1    -7.700, E3 +238886.873}
SPL {X  -165.650, Y  +393.198, Z    +0.000, E1   -17.733, E3 +238885.849}
SPL {X  -165.650, Y  +399.991, Z    +0.000, E1   -27.922, E3 +238886.745}
SPL {X  -165.650, Y  +409.148, Z    +0.000, E1   -43.235, E3 +238882.131}
SPL {X  -165.650, Y  +420.563, Z    +0.000, E1   -54.059, E3 +238882.689}
SPL {X  -165.650, Y  +436.566, Z    +0.000, E1   -62.888, E3 +238884.402}
SPL {X  -165.650, Y  +479.770, Z    +0.000, E1   -67.621, E3 +238903.741}
SPL {X  -165.650, Y  +594.725, Z    +0.000, E1   -69.155, E3 +238971.202}
ENDSPLINE

SPLINE
SPL {X  -165.650, Y  +562.482, Z    +0.000, E1   -62.785, E3 +238990.668}
ENDSPLINE

SPLINE
SPL {X  -165.650, Y  +572.898, Z    +0.000, E1   -62.409, E3 +239004.606}
SPL {X  -165.650, Y  +586.101, Z    +0.000, E1   -62.398, E3 +239018.676}
SPL {X  -165.650, Y  +596.110, Z    +0.000, E1   -62.302, E3 +239030.117}
SPL {X  -165.650, Y  +607.052, Z    +0.000, E1   -62.387, E3 +239041.185}
SPL {X  -165.650, Y  +618.920, Z    +0.000, E1   -62.340, E3 +239054.375}
SPL {X  -165.650, Y  +635.445, Z    +0.000, E1   -62.341, E3 +239072.175}
SPL {X  -165.650, Y  +654.166, Z    +0.000, E1   -62.507, E3 +239091.005}
SPL {X  -165.650, Y  +665.926, Z    +0.000, E1   -62.171, E3 +239105.803}
SPL {X  -165.644, Y  +676.899, Z    +0.000, E1   -62.447, E3 +239115.571}
SPL {X  -165.241, Y  +687.133, Z    +0.000, E1   -62.230, E3 +239128.273}
SPL {X  -164.056, Y  +698.425, Z    +0.000, E1   -62.113, E3 +239141.090}
SPL {X  -162.891, Y  +705.608, Z    +0.000, E1   -61.899, E3 +239150.262}
SPL {X  -160.709, Y  +715.657, Z    +0.000, E1   -61.639, E3 +239163.014}
SPL {X  -157.706, Y  +726.183, Z    +0.000, E1   -61.153, E3 +239177.397}
SPL {X  -155.057, Y  +733.785, Z    +0.000, E1   -60.834, E3 +239187.386}
SPL {X  -152.882, Y  +739.274, Z    +0.000, E1   -60.485, E3 +239195.379}
SPL {X  -149.755, Y  +746.304, Z    +0.000, E1   -59.867, E3 +239206.500}
SPL {X  -146.068, Y  +753.629, Z    +0.000, E1   -59.384, E3 +239216.859}
SPL {X  -143.119, Y  +758.908, Z    +0.000, E1   -58.828, E3 +239225.234}
SPL {X  -141.017, Y  +762.414, Z    +0.000, E1   -58.435, E3 +239230.754}
SPL {X  -132.386, Y  +775.068, Z    +0.000, E1   -61.559, E3 +239229.140}
SPL {X   -89.692, Y  +814.767, Z    +0.000, E1   -54.641, E3 +239343.189}
ENDSPLINE

SPLINE
SPL {X  -133.336, Y  +773.792, Z    +0.000, E1   -47.991, E3 +239471.656}
SPL {X  -153.017, Y  +738.949, Z    +0.000, E1   -37.928, E3 +239485.060}
SPL {X  -160.146, Y  +717.846, Z    +0.000, E1   -27.412, E3 +239472.606}
SPL {X  -163.639, Y  +701.236, Z    +0.000, E1   -18.901, E3 +239478.748}
SPL {X  -165.380, Y  +684.951, Z    +0.000, E1    -8.606, E3 +239477.005}
SPL {X  -165.650, Y  +675.640, Z    +0.000, E1    -1.874, E3 +239476.541}
SPL {X  -165.650, Y  +673.425, Z    +0.000, E1    +0.051, E3 +239475.547}
SPL {X  -165.650, Y  +672.004, Z    +0.000, E1    +1.620, E3 +239475.025}
SPL {X  -165.650, Y  +669.258, Z    +0.000, E1    +5.269, E3 +239474.644}
SPL {X  -165.650, Y  +665.011, Z    +0.000, E1   +11.627, E3 +239474.531}
SPL {X  -165.650, Y  +659.446, Z    +0.000, E1   +21.123, E3 +239473.395}
SPL {X  -165.650, Y  +654.020, Z    +0.000, E1   +29.754, E3 +239473.549}
SPL {X  -165.650, Y  +644.843, Z    +0.000, E1   +43.427, E3 +239471.876}
SPL {X  -165.650, Y  +632.102, Z    +0.000, E1   +56.225, E3 +239471.224}
SPL {X  -165.650, Y  +581.672, Z    +0.000, E1   +69.744, E3 +239483.616}
SPL {X  -165.650, Y  +458.048, Z    +0.000, E1   +68.782, E3 +239564.349}
ENDSPLINE

SPLINE
SPL {X  -165.650, Y  +484.472, Z    +0.000, E1   +63.918, E3 +239578.600}
ENDSPLINE

SPLINE
SPL {X  -165.650, Y  +477.868, Z    +0.000, E1   +63.324, E3 +239589.777}
SPL {X  -165.650, Y  +463.578, Z    +0.000, E1   +63.625, E3 +239602.131}
SPL {X  -165.650, Y  +453.769, Z    +0.000, E1   +63.450, E3 +239613.390}
SPL {X  -165.650, Y  +444.234, Z    +0.000, E1   +63.262, E3 +239624.563}
SPL {X  -165.650, Y  +432.479, Z    +0.000, E1   +63.557, E3 +239634.383}
SPL {X  -165.650, Y  +422.068, Z    +0.000, E1   +63.630, E3 +239644.478}
SPL {X  -165.650, Y  +411.650, Z    +0.000, E1   +63.439, E3 +239656.496}
SPL {X  -165.650, Y  +399.089, Z    +0.000, E1   +63.334, E3 +239670.222}
ENDSPLINE

SPLINE
SPL {X  -165.650, Y  +410.094, Z    +0.000, E1   +60.049, E3 +239680.939}
ENDSPLINE

SPLINE
SPL {X  -165.650, Y  +398.700, Z    +0.000, E1   +60.415, E3 +239691.837}
SPL {X  -165.650, Y  +382.616, Z    +0.000, E1   +61.427, E3 +239703.055}
SPL {X  -165.650, Y  +379.013, Z    +0.000, E1   +60.888, E3 +239710.878}
SPL {X  -165.125, Y  +365.326, Z    +0.000, E1   +61.696, E3 +239720.542}
SPL {X  -164.823, Y  +361.969, Z    +0.000, E1   +60.899, E3 +239729.777}
SPL {X  -163.414, Y  +351.372, Z    +0.000, E1   +61.284, E3 +239739.040}
SPL {X  -162.189, Y  +344.818, Z    +0.000, E1   +60.900, E3 +239748.893}
SPL {X  -160.769, Y  +338.584, Z    +0.000, E1   +60.413, E3 +239759.069}
SPL {X  -157.780, Y  +328.049, Z    +0.000, E1   +60.445, E3 +239770.736}
SPL {X  -155.286, Y  +320.826, Z    +0.000, E1   +59.686, E3 +239783.291}
SPL {X  -152.445, Y  +313.689, Z    +0.000, E1   +59.490, E3 +239792.357}
SPL {X  -150.678, Y  +309.680, Z    +0.000, E1   +58.971, E3 +239799.669}
SPL {X  -148.010, Y  +304.117, Z    +0.000, E1   +58.696, E3 +239807.416}
SPL {X  -144.822, Y  +298.086, Z    +0.000, E1   +58.093, E3 +239817.198}
SPL {X  -142.530, Y  +294.089, Z    +0.000, E1   +57.567, E3 +239824.082}
SPL {X  -136.453, Y  +284.583, Z    +0.000, E1   +60.257, E3 +239821.893}
SPL {X  -128.205, Y  +273.602, Z    +0.000, E1   +62.388, E3 +239822.596}
SPL {X   -96.827, Y  +244.096, Z    +0.000, E1   +56.125, E3 +239901.475}
SPL {X   -90.278, Y  +239.612, Z    +0.000, E1   +54.711, E3 +239931.738}
ENDSPLINE

SPLINE
SPL {X  -110.554, Y  +255.140, Z    +0.000, E1   +52.082, E3 +240041.681}
SPL {X  -144.988, Y  +298.385, Z    +0.000, E1   +42.755, E3 +240065.500}
SPL {X  -160.070, Y  +335.868, Z    +0.000, E1   +27.320, E3 +240062.167}
SPL {X  -163.969, Y  +354.959, Z    +0.000, E1   +17.178, E3 +240062.681}
SPL {X  -165.261, Y  +367.153, Z    +0.000, E1    +9.611, E3 +240061.834}
SPL {X  -165.600, Y  +374.440, Z    +0.000, E1    +4.699, E3 +240061.095}
SPL {X  -165.650, Y  +379.657, Z    +0.000, E1    +0.819, E3 +240060.624}
SPL {X  -165.650, Y  +381.885, Z    +0.000, E1    -1.282, E3 +240059.868}
SPL {X  -165.650, Y  +386.855, Z    +0.000, E1    -7.700, E3 +240059.287}
SPL {X  -165.650, Y  +393.198, Z    +0.000, E1   -17.733, E3 +240058.263}
SPL {X  -165.650, Y  +399.991, Z    +0.000, E1   -27.922, E3 +240059.158}
SPL {X  -165.650, Y  +409.148, Z    +0.000, E1   -43.235, E3 +240054.545}
SPL {X  -165.650, Y  +420.563, Z    +0.000, E1   -54.059, E3 +240055.103}
SPL {X  -165.650, Y  +436.566, Z    +0.000, E1   -62.888, E3 +240056.816}
SPL {X  -165.650, Y  +479.770, Z    +0.000, E1   -67.621, E3 +240076.154}
SPL {X  -165.650, Y  +594.725, Z    +0.000, E1   -69.155, E3 +240143.616}
ENDSPLINE

SPLINE
SPL {X  -165.650, Y  +562.482, Z    +0.000, E1   -62.785, E3 +240163.082}
ENDSPLINE

SPLINE
SPL {X  -165.650, Y  +572.898, Z    +0.000, E1   -62.409, E3 +240177.019}
SPL {X  -165.650, Y  +586.101, Z    +0.000, E1   -62.398, E3 +240191.090}
SPL {X  -165.650, Y  +596.110, Z    +0.000, E1   -62.302, E3 +240202.531}
SPL {X  -165.650, Y  +607.052, Z    +0.000, E1   -62.387, E3 +240213.598}
SPL {X  -165.650, Y  +618.920, Z    +0.000, E1   -62.340, E3 +240226.789}
SPL {X  -165.650, Y  +631.247, Z    +0.000, E1   -62.270, E3 +240240.405}
SPL {X  -165.650, Y  +645.288, Z    +0.000, E1   -62.475, E3 +240254.085}
SPL {X  -165.650, Y  +657.265, Z    +0.000, E1   -62.410, E3 +240267.204}
SPL {X  -165.650, Y  +665.926, Z    +0.000, E1   -62.171, E3 +240278.217}
SPL {X  -165.600, Y  +679.566, Z    +0.000, E1   -62.408, E3 +240291.255}
SPL {X  -165.066, Y  +689.394, Z    +0.000, E1   -62.143, E3 +240303.584}
SPL {X  -164.056, Y  +698.425, Z    +0.000, E1   -62.113, E3 +240313.504}
SPL {X  -162.891, Y  +705.608, Z    +0.000, E1   -61.899, E3 +240322.676}
SPL {X  -161.308, Y  +713.180, Z    +0.000, E1   -61.813, E3 +240331.369}
SPL {X  -159.339, Y  +720.787, Z    +0.000, E1   -61.452, E3 +240342.064}
SPL {X  -156.103, Y  +730.922, Z    +0.000, E1   -60.875, E3 +240356.611}
SPL {X  -152.882, Y  +739.274, Z    +0.000, E1   -60.485, E3 +240367.793}
SPL {X  -150.387, Y  +744.953, Z    +0.000, E1   -60.023, E3 +240376.468}
SPL {X  -147.728, Y  +750.443, Z    +0.000, E1   -59.568, E3 +240384.852}
SPL {X  -143.895, Y  +757.561, Z    +0.000, E1   -58.980, E3 +240395.588}
SPL {X  -141.017, Y  +762.414, Z    +0.000, E1   -58.435, E3 +240403.168}
SPL {X  -134.606, Y  +772.046, Z    +0.000, E1   -61.105, E3 +240400.815}
SPL {X  -127.075, Y  +781.763, Z    +0.000, E1   -62.555, E3 +240403.129}
SPL {X   -89.692, Y  +814.767, Z    +0.000, E1   -54.641, E3 +240515.603}
ENDSPLINE

SPLINE
SPL {X  -133.336, Y  +773.792, Z    +0.000, E1   -47.991, E3 +240644.070}
SPL {X  -153.017, Y  +738.949, Z    +0.000, E1   -37.928, E3 +240657.474}
SPL {X  -160.146, Y  +717.846, Z    +0.000, E1   -27.412, E3 +240645.020}
SPL {X  -163.639, Y  +701.236, Z    +0.000, E1   -18.901, E3 +240651.162}
SPL {X  -165.380, Y  +684.951, Z    +0.000, E1    -8.606, E3 +240649.419}
SPL {X  -165.650, Y  +675.640, Z    +0.000, E1    -1.874, E3 +240648.955}
SPL {X  -165.650, Y  +673.425, Z    +0.000, E1    +0.051, E3 +240647.961}
SPL {X  -165.650, Y  +672.004, Z    +0.000, E1    +1.620, E3 +240647.439}
SPL {X  -165.650, Y  +669.258, Z    +0.000, E1    +5.269, E3 +240647.057}
SPL {X  -165.650, Y  +665.011, Z    +0.000, E1   +11.627, E3 +240646.945}
SPL {X  -165.650, Y  +659.446, Z    +0.000, E1   +21.123, E3 +240645.809}
SPL {X  -165.650, Y  +654.020, Z    +0.000, E1   +29.754, E3 +240645.963}
SPL {X  -165.650, Y  +644.843, Z    +0.000, E1   +43.427, E3 +240644.289}
SPL {X  -165.650, Y  +632.102, Z    +0.000, E1   +56.225, E3 +240643.638}
SPL {X  -165.650, Y  +581.672, Z    +0.000, E1   +69.744, E3 +240656.030}
SPL {X  -165.650, Y  +458.048, Z    +0.000, E1   +68.782, E3 +240736.763}
ENDSPLINE

SPLINE
SPL {X  -165.650, Y  +484.472, Z    +0.000, E1   +63.918, E3 +240751.014}
ENDSPLINE

SPLINE
SPL {X  -165.650, Y  +477.868, Z    +0.000, E1   +63.324, E3 +240762.191}
SPL {X  -165.650, Y  +463.578, Z    +0.000, E1   +63.625, E3 +240774.545}
SPL {X  -165.650, Y  +453.769, Z    +0.000, E1   +63.450, E3 +240785.804}
SPL {X  -165.650, Y  +444.234, Z    +0.000, E1   +63.262, E3 +240796.977}
SPL {X  -165.650, Y  +432.479, Z    +0.000, E1   +63.557, E3 +240806.797}
SPL {X  -165.650, Y  +422.068, Z    +0.000, E1   +63.630, E3 +240816.892}
SPL {X  -165.650, Y  +411.650, Z    +0.000, E1   +63.439, E3 +240828.910}
SPL {X  -165.650, Y  +399.089, Z    +0.000, E1   +63.334, E3 +240842.636}
ENDSPLINE

SPLINE
SPL {X  -165.650, Y  +410.094, Z    +0.000, E1   +60.049, E3 +240853.353}
ENDSPLINE

SPLINE
SPL {X  -165.650, Y  +398.700, Z    +0.000, E1   +60.415, E3 +240864.251}
SPL {X  -165.650, Y  +380.643, Z    +0.000, E1   +61.187, E3 +240879.613}
SPL {X  -165.125, Y  +365.326, Z    +0.000, E1   +61.696, E3 +240892.956}
SPL {X  -164.823, Y  +361.969, Z    +0.000, E1   +60.899, E3 +240902.191}
SPL {X  -163.414, Y  +351.372, Z    +0.000, E1   +61.284, E3 +240911.453}
SPL {X  -162.189, Y  +344.818, Z    +0.000, E1   +60.900, E3 +240921.307}
SPL {X  -160.769, Y  +338.584, Z    +0.000, E1   +60.413, E3 +240931.483}
SPL {X  -157.780, Y  +328.049, Z    +0.000, E1   +60.445, E3 +240943.150}
SPL {X  -155.286, Y  +320.826, Z    +0.000, E1   +59.686, E3 +240955.705}
SPL {X  -152.445, Y  +313.689, Z    +0.000, E1   +59.490, E3 +240964.771}
SPL {X  -149.851, Y  +307.898, Z    +0.000, E1   +58.978, E3 +240974.093}
SPL {X  -146.926, Y  +301.997, Z    +0.000, E1   +58.334, E3 +240984.054}
SPL {X  -143.997, Y  +296.618, Z    +0.000, E1   +58.069, E3 +240991.312}
SPL {X  -142.530, Y  +294.089, Z    +0.000, E1   +57.567, E3 +240996.495}
SPL {X  -134.010, Y  +281.128, Z    +0.000, E1   +60.923, E3 +240994.601}
SPL {X   -93.591, Y  +241.823, Z    +0.000, E1   +55.455, E3 +241087.139}
ENDSPLINE

SPLINE
SPL {X  -110.554, Y  +255.140, Z    +0.000, E1   +52.082, E3 +241214.095}
SPL {X  -137.038, Y  +285.439, Z    +0.000, E1   +46.261, E3 +241233.835}
SPL {X  -149.954, Y  +308.117, Z    +0.000, E1   +39.560, E3 +241240.183}
SPL {X  -160.070, Y  +335.868, Z    +0.000, E1   +27.320, E3 +241234.581}
SPL {X  -163.969, Y  +354.959, Z    +0.000, E1   +17.178, E3 +241235.095}
SPL {X  -165.261, Y  +367.153, Z    +0.000, E1    +9.611, E3 +241234.248}
SPL {X  -165.600, Y  +374.440, Z    +0.000, E1    +4.699, E3 +241233.509}
SPL {X  -165.650, Y  +380.303, Z    +0.000, E1    +0.337, E3 +241232.720}
SPL {X  -165.650, Y  +382.684, Z    +0.000, E1    -2.314, E3 +241232.214}
SPL {X  -165.650, Y  +385.555, Z    +0.000, E1    -6.051, E3 +241231.427}
SPL {X  -165.650, Y  +388.884, Z    +0.000, E1   -10.835, E3 +241232.127}
SPL {X  -165.650, Y  +393.198, Z    +0.000, E1   -17.733, E3 +241230.677}
SPL {X  -165.650, Y  +399.991, Z    +0.000, E1   -27.922, E3 +241231.572}
SPL {X  -165.650, Y  +409.148, Z    +0.000, E1   -43.235, E3 +241226.959}
SPL {X  -165.650, Y  +420.563, Z    +0.000, E1   -54.059, E3 +241227.516}
SPL {X  -165.650, Y  +436.566, Z    +0.000, E1   -62.888, E3 +241229.229}
SPL {X  -165.650, Y  +479.770, Z    +0.000, E1   -67.621, E3 +241248.568}
SPL {X  -165.650, Y  +594.725, Z    +0.000, E1   -69.155, E3 +241316.030}
ENDSPLINE

SPLINE
SPL {X  -165.650, Y  +565.175, Z    +0.000, E1   -62.653, E3 +241339.521}
ENDSPLINE

SPLINE
SPL {X  -165.650, Y  +576.067, Z    +0.000, E1   -62.373, E3 +241352.922}
SPL {X  -165.650, Y  +586.101, Z    +0.000, E1   -62.398, E3 +241363.504}
SPL {X  -165.650, Y  +596.110, Z    +0.000, E1   -62.302, E3 +241374.945}
SPL {X  -165.650, Y  +607.052, Z    +0.000, E1   -62.387, E3 +241386.012}
SPL {X  -165.650, Y  +618.920, Z    +0.000, E1   -62.340, E3 +241399.202}
SPL {X  -165.650, Y  +631.247, Z    +0.000, E1   -62.270, E3 +241412.819}
SPL {X  -165.650, Y  +645.288, Z    +0.000, E1   -62.475, E3 +241426.499}
SPL {X  -165.650, Y  +657.265, Z    +0.000, E1   -62.410, E3 +241439.617}
SPL {X  -165.650, Y  +665.926, Z    +0.000, E1   -62.171, E3 +241450.631}
SPL {X  -165.600, Y  +679.566, Z    +0.000, E1   -62.408, E3 +241463.668}
SPL {X  -165.066, Y  +689.394, Z    +0.000, E1   -62.143, E3 +241475.998}
SPL {X  -164.056, Y  +698.425, Z    +0.000, E1   -62.113, E3 +241485.918}
SPL {X  -162.891, Y  +705.608, Z    +0.000, E1   -61.899, E3 +241495.089}
SPL {X  -160.709, Y  +715.657, Z    +0.000, E1   -61.639, E3 +241507.841}
SPL {X  -157.706, Y  +726.183, Z    +0.000, E1   -61.153, E3 +241522.224}
SPL {X  -155.057, Y  +733.785, Z    +0.000, E1   -60.834, E3 +241532.214}
SPL {X  -152.882, Y  +739.274, Z    +0.000, E1   -60.485, E3 +241540.206}
SPL {X  -150.387, Y  +744.953, Z    +0.000, E1   -60.023, E3 +241548.881}
SPL {X  -146.839, Y  +752.170, Z    +0.000, E1   -59.458, E3 +241559.840}
SPL {X  -142.415, Y  +760.104, Z    +0.000, E1   -58.730, E3 +241571.899}
SPL {X  -132.386, Y  +775.068, Z    +0.000, E1   -61.559, E3 +241573.968}
SPL {X   -89.692, Y  +814.767, Z    +0.000, E1   -54.641, E3 +241688.017}
ENDSPLINE

SPLINE
SPL {X  -133.336, Y  +773.792, Z    +0.000, E1   -47.991, E3 +241816.484}
SPL {X  -153.017, Y  +738.949, Z    +0.000, E1   -37.928, E3 +241829.888}
SPL {X  -160.146, Y  +717.846, Z    +0.000, E1   -27.412, E3 +241817.434}
SPL {X  -163.639, Y  +701.236, Z    +0.000, E1   -18.901, E3 +241823.575}
SPL {X  -165.380, Y  +684.951, Z    +0.000, E1    -8.606, E3 +241821.832}
SPL {X  -165.650, Y  +675.640, Z    +0.000, E1    -1.874, E3 +241821.369}
SPL {X  -165.650, Y  +672.727, Z    +0.000, E1    +0.658, E3 +241820.118}
SPL {X  -165.650, Y  +669.258, Z    +0.000, E1    +5.269, E3 +241819.471}
SPL {X  -165.650, Y  +665.011, Z    +0.000, E1   +11.627, E3 +241819.358}
SPL {X  -165.650, Y  +659.446, Z    +0.000, E1   +21.123, E3 +241818.223}
SPL {X  -165.650, Y  +654.020, Z    +0.000, E1   +29.754, E3 +241818.377}
SPL {X  -165.650, Y  +644.843, Z    +0.000, E1   +43.427, E3 +241816.703}
SPL {X  -165.650, Y  +632.102, Z    +0.000, E1   +56.225, E3 +241816.052}
SPL {X  -165.650, Y  +581.672, Z    +0.000, E1   +69.744, E3 +241828.444}
SPL {X  -165.650, Y  +458.048, Z    +0.000, E1   +68.782, E3 +241909.177}
ENDSPLINE

SPLINE
SPL {X  -165.650, Y  +484.472, Z    +0.000, E1   +63.918, E3 +241923.427}
ENDSPLINE

SPLINE
SPL {X  -165.650, Y  +477.868, Z    +0.000, E1   +63.324, E3 +241934.605}
SPL {X  -165.650, Y  +463.578, Z    +0.000, E1   +63.625, E3 +241946.959}
SPL {X  -165.650, Y  +453.769, Z    +0.000, E1   +63.450, E3 +241958.217}
SPL {X  -165.650, Y  +444.234, Z    +0.000, E1   +63.262, E3 +241969.390}
SPL {X  -165.650, Y  +432.479, Z    +0.000, E1   +63.557, E3 +241979.210}
SPL {X  -165.650, Y  +422.068, Z    +0.000, E1   +63.630, E3 +241989.306}
SPL {X  -165.650, Y  +411.650, Z    +0.000, E1   +63.439, E3 +242001.324}
SPL {X  -165.650, Y  +399.089, Z    +0.000, E1   +63.334, E3 +242015.050}
ENDSPLINE

SPLINE
SPL {X  -165.650, Y  +410.094, Z    +0.000, E1   +60.049, E3 +242025.767}
ENDSPLINE

SPLINE
SPL {X  -165.650, Y  +398.700, Z    +0.000, E1   +60.415, E3 +242036.665}
SPL {X  -165.650, Y  +382.616, Z    +0.000, E1   +61.427, E3 +242047.883}
SPL {X  -165.650, Y  +379.013, Z    +0.000, E1   +60.888, E3 +242055.706}
SPL {X  -165.125, Y  +365.326, Z    +0.000, E1   +61.696, E3 +242065.370}
SPL {X  -164.823, Y  +361.969, Z    +0.000, E1   +60.899, E3 +242074.605}
SPL {X  -163.414, Y  +351.372, Z    +0.000, E1   +61.284, E3 +242083.867}
SPL {X  -162.189, Y  +344.818, Z    +0.000, E1   +60.900, E3 +242093.721}
SPL {X  -160.769, Y  +338.584, Z    +0.000, E1   +60.413, E3 +242103.897}
SPL {X  -158.568, Y  +330.583, Z    +0.000, E1   +60.533, E3 +242112.036}
SPL {X  -157.003, Y  +325.679, Z    +0.000, E1   +60.284, E3 +242119.007}
SPL {X  -155.286, Y  +320.826, Z    +0.000, E1   +59.686, E3 +242128.119}
SPL {X  -152.445, Y  +313.689, Z    +0.000, E1   +59.490, E3 +242137.184}
SPL {X  -150.678, Y  +309.680, Z    +0.000, E1   +58.971, E3 +242144.496}
SPL {X  -148.010, Y  +304.117, Z    +0.000, E1   +58.696, E3 +242152.243}
SPL {X  -144.822, Y  +298.086, Z    +0.000, E1   +58.093, E3 +242162.025}
SPL {X  -142.530, Y  +294.089, Z    +0.000, E1   +57.567, E3 +242168.909}
SPL {X  -134.010, Y  +281.128, Z    +0.000, E1   +60.923, E3 +242167.015}
SPL {X   -93.591, Y  +241.823, Z    +0.000, E1   +55.455, E3 +242259.553}
ENDSPLINE

SPLINE
SPL {X  -110.554, Y  +255.140, Z    +0.000, E1   +52.082, E3 +242386.509}
SPL {X  -137.038, Y  +285.439, Z    +0.000, E1   +46.261, E3 +242406.249}
SPL {X  -149.954, Y  +308.117, Z    +0.000, E1   +39.560, E3 +242412.596}
SPL {X  -160.070, Y  +335.868, Z    +0.000, E1   +27.320, E3 +242406.995}
SPL {X  -163.969, Y  +354.959, Z    +0.000, E1   +17.178, E3 +242407.509}
SPL {X  -165.261, Y  +367.153, Z    +0.000, E1    +9.611, E3 +242406.662}
SPL {X  -165.600, Y  +374.440, Z    +0.000, E1    +4.699, E3 +242405.923}
SPL {X  -165.650, Y  +379.657, Z    +0.000, E1    +0.819, E3 +242405.451}
SPL {X  -165.650, Y  +381.885, Z    +0.000, E1    -1.282, E3 +242404.695}
SPL {X  -165.650, Y  +386.855, Z    +0.000, E1    -7.700, E3 +242404.114}
SPL {X  -165.650, Y  +393.198, Z    +0.000, E1   -17.733, E3 +242403.090}
SPL {X  -165.650, Y  +399.991, Z    +0.000, E1   -27.922, E3 +242403.986}
SPL {X  -165.650, Y  +409.148, Z    +0.000, E1   -43.235, E3 +242399.372}
SPL {X  -165.650, Y  +420.563, Z    +0.000, E1   -54.059, E3 +242399.930}
SPL {X  -165.650, Y  +436.566, Z    +0.000, E1   -62.888, E3 +242401.643}
SPL {X  -165.650, Y  +479.770, Z    +0.000, E1   -67.621, E3 +242420.982}
SPL {X  -165.650, Y  +594.725, Z    +0.000, E1   -69.155, E3 +242488.444}
ENDSPLINE

SPLINE
SPL {X  -165.650, Y  +562.482, Z    +0.000, E1   -62.785, E3 +242507.909}
ENDSPLINE

SPLINE
SPL {X  -165.650, Y  +572.898, Z    +0.000, E1   -62.409, E3 +242521.847}
SPL {X  -165.650, Y  +586.101, Z    +0.000, E1   -62.398, E3 +242535.918}
SPL {X  -165.650, Y  +596.110, Z    +0.000, E1   -62.302, E3 +242547.359}
SPL {X  -165.650, Y  +607.052, Z    +0.000, E1   -62.387, E3 +242558.426}
SPL {X  -165.650, Y  +615.372, Z    +0.000, E1   -62.260, E3 +242568.253}
SPL {X  -165.650, Y  +628.571, Z    +0.000, E1   -62.348, E3 +242581.974}
SPL {X  -165.650, Y  +640.498, Z    +0.000, E1   -62.343, E3 +242594.595}
SPL {X  -165.650, Y  +654.166, Z    +0.000, E1   -62.507, E3 +242608.246}
SPL {X  -165.650, Y  +665.926, Z    +0.000, E1   -62.171, E3 +242623.045}
SPL {X  -165.644, Y  +676.899, Z    +0.000, E1   -62.447, E3 +242632.812}
SPL {X  -165.241, Y  +687.133, Z    +0.000, E1   -62.230, E3 +242645.515}
SPL {X  -164.056, Y  +698.425, Z    +0.000, E1   -62.113, E3 +242658.332}
SPL {X  -162.891, Y  +705.608, Z    +0.000, E1   -61.899, E3 +242667.503}
SPL {X  -160.709, Y  +715.657, Z    +0.000, E1   -61.639, E3 +242680.255}
SPL {X  -157.706, Y  +726.183, Z    +0.000, E1   -61.153, E3 +242694.638}
SPL {X  -155.057, Y  +733.785, Z    +0.000, E1   -60.834, E3 +242704.628}
SPL {X  -152.882, Y  +739.274, Z    +0.000, E1   -60.485, E3 +242712.620}
SPL {X  -150.387, Y  +744.953, Z    +0.000, E1   -60.023, E3 +242721.295}
SPL {X  -146.839, Y  +752.170, Z    +0.000, E1   -59.458, E3 +242732.254}
SPL {X  -142.415, Y  +760.104, Z    +0.000, E1   -58.730, E3 +242744.313}
SPL {X  -134.606, Y  +772.046, Z    +0.000, E1   -61.105, E3 +242745.642}
SPL {X  -127.075, Y  +781.763, Z    +0.000, E1   -62.555, E3 +242747.957}
SPL {X   -89.692, Y  +814.767, Z    +0.000, E1   -54.641, E3 +242860.431}
ENDSPLINE

SPLINE
SPL {X  -133.336, Y  +773.792, Z    +0.000, E1   -47.991, E3 +242988.898}
SPL {X  -153.017, Y  +738.949, Z    +0.000, E1   -37.928, E3 +243002.301}
SPL {X  -160.146, Y  +717.846, Z    +0.000, E1   -27.412, E3 +242989.848}
SPL {X  -163.639, Y  +701.236, Z    +0.000, E1   -18.901, E3 +242995.989}
SPL {X  -165.380, Y  +684.951, Z    +0.000, E1    -8.606, E3 +242994.246}
SPL {X  -165.650, Y  +675.640, Z    +0.000, E1    -1.874, E3 +242993.782}
SPL {X  -165.650, Y  +673.425, Z    +0.000, E1    +0.051, E3 +242992.788}
SPL {X  -165.650, Y  +672.004, Z    +0.000, E1    +1.620, E3 +242992.267}
SPL {X  -165.650, Y  +669.258, Z    +0.000, E1    +5.269, E3 +242991.885}
SPL {X  -165.650, Y  +665.011, Z    +0.000, E1   +11.627, E3 +242991.772}
SPL {X  -165.650, Y  +659.446, Z    +0.000, E1   +21.123, E3 +242990.636}
SPL {X  -165.650, Y  +651.038, Z    +0.000, E1   +34.281, E3 +242990.262}
SPL {X  -165.650, Y  +635.255, Z    +0.000, E1   +53.641, E3 +242988.450}
SPL {X  -165.650, Y  +581.672, Z    +0.000, E1   +69.744, E3 +243000.858}
SPL {X  -165.650, Y  +458.048, Z    +0.000, E1   +68.782, E3 +243081.591}
ENDSPLINE

SPLINE
SPL {X  -165.650, Y  +484.472, Z    +0.000, E1   +63.918, E3 +243095.841}
ENDSPLINE

SPLINE
SPL {X  -165.650, Y  +477.868, Z    +0.000, E1   +63.324, E3 +243107.019}
SPL {X  -165.650, Y  +463.578, Z    +0.000, E1   +63.625, E3 +243119.373}
SPL {X  -165.650, Y  +453.769, Z    +0.000, E1   +63.450, E3 +243130.631}
SPL {X  -165.650, Y  +444.234, Z    +0.000, E1   +63.262, E3 +243141.804}
SPL {X  -165.650, Y  +432.479, Z    +0.000, E1   +63.557, E3 +243151.624}
SPL {X  -165.650, Y  +422.068, Z    +0.000, E1   +63.630, E3 +243161.719}
SPL {X  -165.650, Y  +409.231, Z    +0.000, E1   +63.364, E3 +243176.968}
SPL {X  -165.650, Y  +395.008, Z    +0.000, E1   +63.445, E3 +243190.731}
ENDSPLINE

SPLINE
SPL {X  -165.650, Y  +410.094, Z    +0.000, E1   +60.049, E3 +243198.181}
ENDSPLINE

SPLINE
SPL {X  -165.650, Y  +398.700, Z    +0.000, E1   +60.415, E3 +243209.079}
SPL {X  -165.650, Y  +382.616, Z    +0.000, E1   +61.427, E3 +243220.297}
SPL {X  -165.650, Y  +379.013, Z    +0.000, E1   +60.888, E3 +243228.120}
SPL {X  -165.125, Y  +365.326, Z    +0.000, E1   +61.696, E3 +243237.784}
SPL {X  -164.823, Y  +361.969, Z    +0.000, E1   +60.899, E3 +243247.019}
SPL {X  -163.414, Y  +351.372, Z    +0.000, E1   +61.284, E3 +243256.281}
SPL {X  -162.189, Y  +344.818, Z    +0.000, E1   +60.900, E3 +243266.134}
SPL {X  -160.769, Y  +338.584, Z    +0.000, E1   +60.413, E3 +243276.310}
SPL {X  -157.780, Y  +328.049, Z    +0.000, E1   +60.445, E3 +243287.977}
SPL {X  -155.286, Y  +320.826, Z    +0.000, E1   +59.686, E3 +243300.533}
SPL {X  -152.445, Y  +313.689, Z    +0.000, E1   +59.490, E3 +243309.598}
SPL {X  -150.678, Y  +309.680, Z    +0.000, E1   +58.971, E3 +243316.910}
SPL {X  -148.010, Y  +304.117, Z    +0.000, E1   +58.696, E3 +243324.657}
SPL {X  -144.822, Y  +298.086, Z    +0.000, E1   +58.093, E3 +243334.439}
SPL {X  -142.530, Y  +294.089, Z    +0.000, E1   +57.567, E3 +243341.323}
SPL {X  -136.453, Y  +284.583, Z    +0.000, E1   +60.257, E3 +243339.134}
SPL {X  -128.205, Y  +273.602, Z    +0.000, E1   +62.388, E3 +243339.837}
SPL {X   -93.591, Y  +241.823, Z    +0.000, E1   +55.455, E3 +243431.967}
ENDSPLINE

SPLINE
SPL {X  -110.554, Y  +255.140, Z    +0.000, E1   +52.082, E3 +243558.923}
SPL {X  -137.038, Y  +285.439, Z    +0.000, E1   +46.261, E3 +243578.662}
SPL {X  -149.954, Y  +308.117, Z    +0.000, E1   +39.560, E3 +243585.010}
SPL {X  -160.070, Y  +335.868, Z    +0.000, E1   +27.320, E3 +243579.409}
SPL {X  -163.969, Y  +354.959, Z    +0.000, E1   +17.178, E3 +243579.923}
SPL {X  -165.261, Y  +367.153, Z    +0.000, E1    +9.611, E3 +243579.075}
SPL {X  -165.600, Y  +374.440, Z    +0.000, E1    +4.699, E3 +243578.337}
SPL {X  -165.650, Y  +379.657, Z    +0.000, E1    +0.819, E3 +243577.865}
SPL {X  -165.650, Y  +381.885, Z    +0.000, E1    -1.282, E3 +243577.109}
SPL {X  -165.650, Y  +386.855, Z    +0.000, E1    -7.700, E3 +243576.528}
SPL {X  -165.650, Y  +393.198, Z    +0.000, E1   -17.733, E3 +243575.504}
SPL {X  -165.650, Y  +399.991, Z    +0.000, E1   -27.922, E3 +243576.400}
SPL {X  -165.650, Y  +409.148, Z    +0.000, E1   -43.235, E3 +243571.786}
SPL {X  -165.650, Y  +420.563, Z    +0.000, E1   -54.059, E3 +243572.344}
SPL {X  -165.650, Y  +436.566, Z    +0.000, E1   -62.888, E3 +243574.057}
SPL {X  -165.650, Y  +479.770, Z    +0.000, E1   -67.621, E3 +243593.396}
SPL {X  -165.650, Y  +594.725, Z    +0.000, E1   -69.155, E3 +243660.858}
ENDSPLINE

SPLINE
SPL {X  -165.650, Y  +562.482, Z    +0.000, E1   -62.785, E3 +243680.323}
ENDSPLINE

SPLINE
SPL {X  -165.650, Y  +572.898, Z    +0.000, E1   -62.409, E3 +243694.261}
SPL {X  -165.650, Y  +586.101, Z    +0.000, E1   -62.398, E3 +243708.332}
SPL {X  -165.650, Y  +596.110, Z    +0.000, E1   -62.302, E3 +243719.773}
SPL {X  -165.650, Y  +607.052, Z    +0.000, E1   -62.387, E3 +243730.840}
SPL {X  -165.650, Y  +618.920, Z    +0.000, E1   -62.340, E3 +243744.030}
SPL {X  -165.650, Y  +635.445, Z    +0.000, E1   -62.341, E3 +243761.831}
SPL {X  -165.650, Y  +654.166, Z    +0.000, E1   -62.507, E3 +243780.660}
SPL {X  -165.650, Y  +665.926, Z    +0.000, E1   -62.171, E3 +243795.459}
SPL {X  -165.644, Y  +676.899, Z    +0.000, E1   -62.447, E3 +243805.226}
SPL {X  -165.241, Y  +687.133, Z    +0.000, E1   -62.230, E3 +243817.929}
SPL {X  -164.056, Y  +698.425, Z    +0.000, E1   -62.113, E3 +243830.745}
SPL {X  -162.891, Y  +705.608, Z    +0.000, E1   -61.899, E3 +243839.917}
SPL {X  -160.709, Y  +715.657, Z    +0.000, E1   -61.639, E3 +243852.669}
SPL {X  -157.706, Y  +726.183, Z    +0.000, E1   -61.153, E3 +243867.052}
SPL {X  -155.057, Y  +733.785, Z    +0.000, E1   -60.834, E3 +243877.041}
SPL {X  -152.882, Y  +739.274, Z    +0.000, E1   -60.485, E3 +243885.034}
SPL {X  -149.755, Y  +746.304, Z    +0.000, E1   -59.867, E3 +243896.155}
SPL {X  -146.068, Y  +753.629, Z    +0.000, E1   -59.384, E3 +243906.515}
SPL {X  -143.119, Y  +758.908, Z    +0.000, E1   -58.828, E3 +243914.889}
SPL {X  -141.017, Y  +762.414, Z    +0.000, E1   -58.435, E3 +243920.410}
SPL {X  -134.606, Y  +772.046, Z    +0.000, E1   -61.105, E3 +243918.056}
SPL {X  -127.075, Y  +781.763, Z    +0.000, E1   -62.555, E3 +243920.370}
SPL {X   -95.057, Y  +811.161, Z    +0.000, E1   -56.196, E3 +244000.424}
SPL {X   -88.361, Y  +815.615, Z    +0.000, E1   -54.176, E3 +244046.341}
ENDSPLINE

SPLINE
SPL {X  -120.253, Y  +789.426, Z    +0.000, E1   -51.165, E3 +244154.119}
SPL {X  -143.101, Y  +758.939, Z    +0.000, E1   -44.365, E3 +244168.226}
SPL {X  -158.740, Y  +722.846, Z    +0.000, E1   -30.140, E3 +244166.265}
SPL {X  -163.639, Y  +701.236, Z    +0.000, E1   -18.901, E3 +244168.403}
SPL {X  -165.058, Y  +689.494, Z    +0.000, E1   -11.557, E3 +244167.220}
SPL {X  -165.574, Y  +680.514, Z    +0.000, E1    -5.500, E3 +244166.464}
SPL {X  -165.650, Y  +673.883, Z    +0.000, E1    -0.454, E3 +244165.475}
SPL {X  -165.650, Y  +672.004, Z    +0.000, E1    +1.620, E3 +244164.681}
SPL {X  -165.650, Y  +669.258, Z    +0.000, E1    +5.269, E3 +244164.299}
SPL {X  -165.650, Y  +665.011, Z    +0.000, E1   +11.627, E3 +244164.186}
SPL {X  -165.650, Y  +659.446, Z    +0.000, E1   +21.123, E3 +244163.050}
SPL {X  -165.650, Y  +651.038, Z    +0.000, E1   +34.281, E3 +244162.676}
SPL {X  -165.650, Y  +635.255, Z    +0.000, E1   +53.641, E3 +244160.864}
SPL {X  -165.650, Y  +581.672, Z    +0.000, E1   +69.744, E3 +244173.272}
SPL {X  -165.650, Y  +458.048, Z    +0.000, E1   +68.782, E3 +244254.004}
ENDSPLINE

SPLINE
SPL {X  -165.650, Y  +484.472, Z    +0.000, E1   +63.918, E3 +244268.255}
ENDSPLINE

SPLINE
SPL {X  -165.650, Y  +477.868, Z    +0.000, E1   +63.324, E3 +244279.433}
SPL {X  -165.650, Y  +463.578, Z    +0.000, E1   +63.625, E3 +244291.786}
SPL {X  -165.650, Y  +453.769, Z    +0.000, E1   +63.450, E3 +244303.045}
SPL {X  -165.650, Y  +444.234, Z    +0.000, E1   +63.262, E3 +244314.218}
SPL {X  -165.650, Y  +432.479, Z    +0.000, E1   +63.557, E3 +244324.038}
SPL {X  -165.650, Y  +422.068, Z    +0.000, E1   +63.630, E3 +244334.133}
SPL {X  -165.650, Y  +409.231, Z    +0.000, E1   +63.364, E3 +244349.382}
SPL {X  -165.650, Y  +395.008, Z    +0.000, E1   +63.445, E3 +244363.145}
ENDSPLINE

SPLINE
SPL {X  -165.650, Y  +410.094, Z    +0.000, E1   +60.049, E3 +244370.594}
ENDSPLINE

SPLINE
SPL {X  -165.650, Y  +398.700, Z    +0.000, E1   +60.415, E3 +244381.492}
SPL {X  -165.650, Y  +383.349, Z    +0.000, E1   +61.276, E3 +244392.993}
ENDSPLINE

SPLINE
SPL {X  -165.650, Y  +398.905, Z    +0.000, E1   +57.332, E3 +244400.737}
ENDSPLINE

SPLINE
SPL {X  -165.650, Y  +388.492, Z    +0.000, E1   +57.709, E3 +244411.854}
SPL {X  -165.650, Y  +379.894, Z    +0.000, E1   +57.709, E3 +244422.958}
SPL {X  -165.538, Y  +372.423, Z    +0.000, E1   +57.528, E3 +244433.831}
SPL {X  -164.865, Y  +362.388, Z    +0.000, E1   +57.628, E3 +244446.218}
SPL {X  -163.867, Y  +354.258, Z    +0.000, E1   +57.359, E3 +244458.435}
SPL {X  -162.678, Y  +347.264, Z    +0.000, E1   +57.150, E3 +244468.776}
SPL {X  -161.618, Y  +342.173, Z    +0.000, E1   +56.783, E3 +244477.661}
SPL {X  -159.878, Y  +335.155, Z    +0.000, E1   +56.685, E3 +244487.465}
SPL {X  -158.009, Y  +328.771, Z    +0.000, E1   +56.325, E3 +244497.825}
SPL {X  -156.065, Y  +322.971, Z    +0.000, E1   +56.177, E3 +244506.169}
SPL {X  -154.487, Y  +318.719, Z    +0.000, E1   +55.733, E3 +244514.177}
SPL {X  -151.902, Y  +312.426, Z    +0.000, E1   +55.494, E3 +244523.652}
SPL {X  -149.742, Y  +307.668, Z    +0.000, E1   +54.896, E3 +244532.864}
SPL {X  -146.487, Y  +301.160, Z    +0.000, E1   +54.808, E3 +244541.727}
SPL {X  -133.590, Y  +280.553, Z    +0.000, E1   +59.642, E3 +244542.684}
SPL {X  -112.638, Y  +257.040, Z    +0.000, E1   +51.417, E3 +244646.067}
ENDSPLINE

SPLINE
SPL {X  -115.209, Y  +259.476, Z    +0.000, E1   +49.595, E3 +244679.338}
SPL {X  -147.344, Y  +302.806, Z    +0.000, E1   +40.158, E3 +244768.800}
SPL {X  -160.798, Y  +338.700, Z    +0.000, E1   +25.294, E3 +244768.282}
SPL {X  -163.893, Y  +354.439, Z    +0.000, E1   +16.805, E3 +244762.756}
SPL {X  -165.158, Y  +365.746, Z    +0.000, E1   +10.198, E3 +244760.699}
SPL {X  -165.639, Y  +376.620, Z    +0.000, E1    +3.186, E3 +244760.499}
SPL {X  -165.650, Y  +381.477, Z    +0.000, E1    -0.622, E3 +244759.309}
SPL {X  -165.650, Y  +384.861, Z    +0.000, E1    -4.465, E3 +244758.712}
SPL {X  -165.650, Y  +388.792, Z    +0.000, E1    -9.482, E3 +244758.028}
SPL {X  -165.650, Y  +393.970, Z    +0.000, E1   -17.146, E3 +244757.184}
SPL {X  -165.650, Y  +401.614, Z    +0.000, E1   -27.619, E3 +244757.839}
SPL {X  -165.650, Y  +418.105, Z    +0.000, E1   -49.413, E3 +244753.247}
SPL {X  -165.650, Y  +465.736, Z    +0.000, E1   -65.678, E3 +244766.990}
SPL {X  -165.650, Y  +519.483, Z    +0.000, E1   -68.357, E3 +244793.175}
SPL {X  -165.650, Y  +548.869, Z    +0.000, E1   -62.199, E3 +244848.867}
ENDSPLINE

SPLINE
SPL {X  -165.650, Y  +534.780, Z    +0.000, E1   -57.803, E3 +244862.517}
ENDSPLINE

SPLINE
SPL {X  -165.650, Y  +545.905, Z    +0.000, E1   -57.853, E3 +244876.456}
SPL {X  -165.650, Y  +553.630, Z    +0.000, E1   -57.616, E3 +244887.906}
SPL {X  -165.650, Y  +563.473, Z    +0.000, E1   -57.690, E3 +244900.270}
SPL {X  -165.650, Y  +573.011, Z    +0.000, E1   -57.610, E3 +244913.061}
SPL {X  -165.650, Y  +581.530, Z    +0.000, E1   -57.678, E3 +244923.659}
SPL {X  -165.650, Y  +589.475, Z    +0.000, E1   -57.572, E3 +244934.646}
SPL {X  -165.650, Y  +599.695, Z    +0.000, E1   -57.964, E3 +244945.262}
SPL {X  -165.650, Y  +606.915, Z    +0.000, E1   -57.651, E3 +244956.619}
SPL {X  -165.650, Y  +614.927, Z    +0.000, E1   -57.517, E3 +244967.888}
SPL {X  -165.650, Y  +624.337, Z    +0.000, E1   -57.671, E3 +244979.114}
SPL {X  -165.650, Y  +634.236, Z    +0.000, E1   -57.671, E3 +244991.965}
SPL {X  -165.650, Y  +644.287, Z    +0.000, E1   -57.872, E3 +245003.531}
SPL {X  -165.650, Y  +650.480, Z    +0.000, E1   -57.669, E3 +245012.836}
SPL {X  -165.650, Y  +657.986, Z    +0.000, E1   -57.646, E3 +245022.728}
SPL {X  -165.650, Y  +667.585, Z    +0.000, E1   -57.803, E3 +245034.123}
SPL {X  -165.650, Y  +673.199, Z    +0.000, E1   -57.412, E3 +245043.867}
SPL {X  -165.558, Y  +681.013, Z    +0.000, E1   -57.768, E3 +245051.707}
SPL {X  -165.167, Y  +688.139, Z    +0.000, E1   -57.463, E3 +245063.005}
SPL {X  -164.323, Y  +696.426, Z    +0.000, E1   -57.565, E3 +245072.992}
SPL {X  -163.313, Y  +703.224, Z    +0.000, E1   -57.403, E3 +245082.886}
SPL {X  -161.906, Y  +710.520, Z    +0.000, E1   -57.149, E3 +245093.837}
SPL {X  -160.577, Y  +716.182, Z    +0.000, E1   -56.676, E3 +245104.098}
SPL {X  -158.520, Y  +723.576, Z    +0.000, E1   -56.758, E3 +245113.143}
SPL {X  -156.858, Y  +728.749, Z    +0.000, E1   -56.333, E3 +245122.285}
SPL {X  -155.155, Y  +733.525, Z    +0.000, E1   -55.869, E3 +245131.062}
SPL {X  -152.530, Y  +740.111, Z    +0.000, E1   -55.545, E3 +245141.538}
SPL {X  -149.057, Y  +747.763, Z    +0.000, E1   -54.897, E3 +245154.743}
SPL {X  -146.339, Y  +753.120, Z    +0.000, E1   -54.477, E3 +245163.628}
SPL {X  -137.656, Y  +767.645, Z    +0.000, E1   -58.229, E3 +245163.338}
SPL {X  -110.324, Y  +799.066, Z    +0.000, E1   -54.396, E3 +245232.874}
SPL {X  -100.308, Y  +807.326, Z    +0.000, E1   -52.880, E3 +245277.441}
ENDSPLINE

SPLINE
SPL {X  -108.196, Y  +800.934, Z    +0.000, E1   -52.068, E3 +245369.768}
SPL {X  -144.673, Y  +756.182, Z    +0.000, E1   -41.752, E3 +245387.846}
SPL {X  -160.601, Y  +716.087, Z    +0.000, E1   -25.730, E3 +245387.474}
SPL {X  -164.850, Y  +691.761, Z    +0.000, E1   -12.424, E3 +245384.741}
SPL {X  -165.596, Y  +679.730, Z    +0.000, E1    -4.777, E3 +245383.615}
SPL {X  -165.650, Y  +674.376, Z    +0.000, E1    -0.866, E3 +245383.530}
SPL {X  -165.650, Y  +672.384, Z    +0.000, E1    +0.908, E3 +245382.411}
SPL {X  -165.650, Y  +669.968, Z    +0.000, E1    +3.584, E3 +245382.227}
SPL {X  -165.650, Y  +666.667, Z    +0.000, E1    +7.761, E3 +245381.907}
SPL {X  -165.650, Y  +662.028, Z    +0.000, E1   +14.359, E3 +245381.537}
SPL {X  -165.650, Y  +654.885, Z    +0.000, E1   +25.204, E3 +245380.052}
SPL {X  -165.650, Y  +641.882, Z    +0.000, E1   +46.566, E3 +245372.923}
SPL {X  -165.650, Y  +630.946, Z    +0.000, E1   +55.779, E3 +245373.598}
SPL {X  -165.650, Y  +590.135, Z    +0.000, E1   +59.110, E3 +245406.217}
SPL {X  -165.650, Y  +491.251, Z    +0.000, E1   +65.373, E3 +245465.647}
ENDSPLINE

SPLINE
SPL {X  -165.650, Y  +517.534, Z    +0.000, E1   +59.090, E3 +245480.244}
ENDSPLINE

SPLINE
SPL {X  -165.650, Y  +515.821, Z    +0.000, E1   +58.153, E3 +245488.692}
SPL {X  -165.650, Y  +506.715, Z    +0.000, E1   +58.090, E3 +245500.780}
SPL {X  -165.650, Y  +496.085, Z    +0.000, E1   +57.984, E3 +245515.028}
SPL {X  -165.650, Y  +485.167, Z    +0.000, E1   +58.003, E3 +245528.859}
ENDSPLINE

SPLINE
SPL {X  -165.650, Y  +505.180, Z    +0.000, E1   +52.333, E3 +245535.612}
SPL {X  -165.650, Y  +506.534, Z    +0.000, E1   +50.148, E3 +245547.071}
ENDSPLINE

SPLINE
SPL {X  -165.650, Y  +495.166, Z    +0.000, E1   +51.070, E3 +245560.499}
SPL {X  -165.650, Y  +485.807, Z    +0.000, E1   +51.973, E3 +245570.232}
SPL {X  -165.650, Y  +478.030, Z    +0.000, E1   +52.389, E3 +245580.039}
SPL {X  -165.650, Y  +467.527, Z    +0.000, E1   +53.334, E3 +245590.533}
SPL {X  -165.650, Y  +453.744, Z    +0.000, E1   +54.190, E3 +245606.014}
SPL {X  -165.650, Y  +440.843, Z    +0.000, E1   +55.023, E3 +245619.435}
SPL {X  -165.650, Y  +431.771, Z    +0.000, E1   +55.549, E3 +245628.952}
SPL {X  -165.650, Y  +420.799, Z    +0.000, E1   +56.452, E3 +245638.338}
SPL {X  -165.650, Y  +409.731, Z    +0.000, E1   +57.273, E3 +245647.826}
SPL {X  -165.650, Y  +399.687, Z    +0.000, E1   +57.433, E3 +245660.011}
SPL {X  -165.650, Y  +388.492, Z    +0.000, E1   +57.709, E3 +245672.724}
SPL {X  -165.650, Y  +379.894, Z    +0.000, E1   +57.709, E3 +245683.828}
SPL {X  -165.399, Y  +369.388, Z    +0.000, E1   +57.657, E3 +245697.922}
SPL {X  -164.717, Y  +360.945, Z    +0.000, E1   +57.468, E3 +245709.859}
SPL {X  -163.867, Y  +354.258, Z    +0.000, E1   +57.359, E3 +245719.304}
SPL {X  -162.678, Y  +347.264, Z    +0.000, E1   +57.150, E3 +245729.645}
SPL {X  -161.618, Y  +342.173, Z    +0.000, E1   +56.783, E3 +245738.531}
SPL {X  -159.878, Y  +335.155, Z    +0.000, E1   +56.685, E3 +245748.335}
SPL {X  -158.009, Y  +328.771, Z    +0.000, E1   +56.325, E3 +245758.694}
SPL {X  -156.065, Y  +322.971, Z    +0.000, E1   +56.177, E3 +245767.038}
SPL {X  -153.731, Y  +316.803, Z    +0.000, E1   +55.737, E3 +245777.614}
SPL {X  -150.320, Y  +308.902, Z    +0.000, E1   +55.085, E3 +245791.311}
SPL {X  -147.957, Y  +304.011, Z    +0.000, E1   +54.431, E3 +245800.773}
SPL {X  -144.791, Y  +298.030, Z    +0.000, E1   +55.214, E3 +245804.631}
SPL {X  -133.590, Y  +280.553, Z    +0.000, E1   +59.642, E3 +245803.554}
SPL {X  -112.638, Y  +257.040, Z    +0.000, E1   +51.417, E3 +245906.937}
ENDSPLINE

SPLINE
SPL {X  -115.209, Y  +259.476, Z    +0.000, E1   +49.595, E3 +245940.207}
SPL {X  -147.344, Y  +302.806, Z    +0.000, E1   +40.158, E3 +246029.669}
SPL {X  -160.798, Y  +338.700, Z    +0.000, E1   +25.294, E3 +246029.151}
SPL {X  -163.893, Y  +354.439, Z    +0.000, E1   +16.805, E3 +246023.625}
SPL {X  -165.158, Y  +365.746, Z    +0.000, E1   +10.198, E3 +246021.568}
SPL {X  -165.639, Y  +376.620, Z    +0.000, E1    +3.186, E3 +246021.368}
SPL {X  -165.650, Y  +380.533, Z    +0.000, E1    +0.120, E3 +246020.396}
SPL {X  -165.650, Y  +383.454, Z    +0.000, E1    -2.667, E3 +246019.803}
SPL {X  -165.650, Y  +388.792, Z    +0.000, E1    -9.482, E3 +246018.897}
SPL {X  -165.650, Y  +396.421, Z    +0.000, E1   -20.352, E3 +246018.695}
SPL {X  -165.650, Y  +404.249, Z    +0.000, E1   -31.650, E3 +246018.074}
SPL {X  -165.650, Y  +418.105, Z    +0.000, E1   -49.413, E3 +246014.117}
SPL {X  -165.650, Y  +465.736, Z    +0.000, E1   -65.678, E3 +246027.859}
SPL {X  -165.650, Y  +519.483, Z    +0.000, E1   -68.357, E3 +246054.044}
SPL {X  -165.650, Y  +548.869, Z    +0.000, E1   -62.199, E3 +246109.737}
ENDSPLINE

SPLINE
SPL {X  -165.650, Y  +530.735, Z    +0.000, E1   -57.778, E3 +246118.161}
ENDSPLINE

SPLINE
SPL {X  -165.650, Y  +536.777, Z    +0.000, E1   -57.774, E3 +246126.038}
SPL {X  -165.650, Y  +545.905, Z    +0.000, E1   -57.853, E3 +246137.326}
SPL {X  -165.650, Y  +553.630, Z    +0.000, E1   -57.616, E3 +246148.775}
SPL {X  -165.650, Y  +563.473, Z    +0.000, E1   -57.690, E3 +246161.139}
SPL {X  -165.650, Y  +573.011, Z    +0.000, E1   -57.610, E3 +246173.930}
SPL {X  -165.650, Y  +581.530, Z    +0.000, E1   -57.678, E3 +246184.528}
SPL {X  -165.650, Y  +589.475, Z    +0.000, E1   -57.572, E3 +246195.515}
SPL {X  -165.650, Y  +599.695, Z    +0.000, E1   -57.964, E3 +246206.132}
SPL {X  -165.650, Y  +606.915, Z    +0.000, E1   -57.651, E3 +246217.488}
SPL {X  -165.650, Y  +614.927, Z    +0.000, E1   -57.517, E3 +246228.758}
SPL {X  -165.650, Y  +624.337, Z    +0.000, E1   -57.671, E3 +246239.984}
SPL {X  -165.650, Y  +634.236, Z    +0.000, E1   -57.671, E3 +246252.834}
SPL {X  -165.650, Y  +644.287, Z    +0.000, E1   -57.872, E3 +246264.400}
SPL {X  -165.650, Y  +650.480, Z    +0.000, E1   -57.669, E3 +246273.705}
SPL {X  -165.650, Y  +657.986, Z    +0.000, E1   -57.646, E3 +246283.597}
SPL {X  -165.650, Y  +667.585, Z    +0.000, E1   -57.803, E3 +246294.993}
SPL {X  -165.634, Y  +677.794, Z    +0.000, E1   -57.650, E3 +246309.295}
SPL {X  -165.167, Y  +688.139, Z    +0.000, E1   -57.463, E3 +246323.874}
SPL {X  -164.323, Y  +696.426, Z    +0.000, E1   -57.565, E3 +246333.861}
SPL {X  -163.313, Y  +703.224, Z    +0.000, E1   -57.403, E3 +246343.755}
SPL {X  -161.906, Y  +710.520, Z    +0.000, E1   -57.149, E3 +246354.706}
SPL {X  -160.577, Y  +716.182, Z    +0.000, E1   -56.676, E3 +246364.967}
SPL {X  -158.520, Y  +723.576, Z    +0.000, E1   -56.758, E3 +246374.012}
SPL {X  -156.858, Y  +728.749, Z    +0.000, E1   -56.333, E3 +246383.155}
SPL {X  -155.155, Y  +733.525, Z    +0.000, E1   -55.869, E3 +246391.931}
SPL {X  -153.442, Y  +737.914, Z    +0.000, E1   -55.562, E3 +246399.336}
SPL {X  -150.574, Y  +744.547, Z    +0.000, E1   -55.310, E3 +246409.319}
SPL {X  -147.713, Y  +750.471, Z    +0.000, E1   -54.514, E3 +246420.981}
SPL {X  -139.786, Y  +764.381, Z    +0.000, E1   -57.209, E3 +246425.169}
SPL {X  -110.324, Y  +799.066, Z    +0.000, E1   -54.396, E3 +246493.743}
SPL {X  -100.308, Y  +807.326, Z    +0.000, E1   -52.880, E3 +246538.311}
ENDSPLINE

SPLINE
SPL {X  -108.196, Y  +800.934, Z    +0.000, E1   -52.068, E3 +246630.637}
SPL {X  -147.753, Y  +750.393, Z    +0.000, E1   -39.863, E3 +246648.860}
SPL {X  -161.414, Y  +712.720, Z    +0.000, E1   -24.024, E3 +246648.202}
SPL {X  -164.278, Y  +696.774, Z    +0.000, E1   -15.225, E3 +246642.813}
SPL {X  -165.078, Y  +689.251, Z    +0.000, E1   -10.876, E3 +246646.966}
SPL {X  -165.596, Y  +679.730, Z    +0.000, E1    -4.777, E3 +246644.485}
SPL {X  -165.650, Y  +674.376, Z    +0.000, E1    -0.866, E3 +246644.400}
SPL {X  -165.650, Y  +672.384, Z    +0.000, E1    +0.908, E3 +246643.281}
SPL {X  -165.650, Y  +669.968, Z    +0.000, E1    +3.584, E3 +246643.097}
SPL {X  -165.650, Y  +666.667, Z    +0.000, E1    +7.761, E3 +246642.776}
SPL {X  -165.650, Y  +662.028, Z    +0.000, E1   +14.359, E3 +246642.406}
SPL {X  -165.650, Y  +654.885, Z    +0.000, E1   +25.204, E3 +246640.921}
SPL {X  -165.650, Y  +641.882, Z    +0.000, E1   +46.566, E3 +246633.793}
SPL {X  -165.650, Y  +630.946, Z    +0.000, E1   +55.779, E3 +246634.467}
SPL {X  -165.650, Y  +590.135, Z    +0.000, E1   +59.110, E3 +246667.087}
SPL {X  -165.650, Y  +491.251, Z    +0.000, E1   +65.373, E3 +246726.516}
ENDSPLINE

SPLINE
SPL {X  -165.650, Y  +514.386, Z    +0.000, E1   +58.403, E3 +246750.066}
ENDSPLINE

SPLINE
SPL {X  -165.650, Y  +502.532, Z    +0.000, E1   +57.988, E3 +246767.682}
SPL {X  -165.650, Y  +493.307, Z    +0.000, E1   +58.045, E3 +246778.951}
SPL {X  -165.650, Y  +485.167, Z    +0.000, E1   +58.003, E3 +246789.729}
ENDSPLINE

SPLINE
SPL {X  -165.650, Y  +509.193, Z    +0.000, E1   +50.604, E3 +246800.696}
ENDSPLINE

SPLINE
SPL {X  -165.650, Y  +503.302, Z    +0.000, E1   +50.402, E3 +246811.792}
SPL {X  -165.650, Y  +495.166, Z    +0.000, E1   +51.070, E3 +246821.369}
SPL {X  -165.650, Y  +485.807, Z    +0.000, E1   +51.973, E3 +246831.102}
SPL {X  -165.650, Y  +478.030, Z    +0.000, E1   +52.389, E3 +246840.909}
SPL {X  -165.650, Y  +467.527, Z    +0.000, E1   +53.334, E3 +246851.403}
SPL {X  -165.650, Y  +457.379, Z    +0.000, E1   +53.935, E3 +246862.946}
SPL {X  -165.650, Y  +444.120, Z    +0.000, E1   +54.815, E3 +246876.992}
SPL {X  -165.650, Y  +431.771, Z    +0.000, E1   +55.549, E3 +246889.822}
SPL {X  -165.650, Y  +420.799, Z    +0.000, E1   +56.452, E3 +246899.208}
SPL {X  -165.650, Y  +409.731, Z    +0.000, E1   +57.273, E3 +246908.696}
SPL {X  -165.650, Y  +399.687, Z    +0.000, E1   +57.433, E3 +246920.880}
SPL {X  -165.650, Y  +388.492, Z    +0.000, E1   +57.709, E3 +246933.594}
SPL {X  -165.650, Y  +379.894, Z    +0.000, E1   +57.709, E3 +246944.697}
SPL {X  -165.538, Y  +372.423, Z    +0.000, E1   +57.528, E3 +246955.570}
SPL {X  -164.865, Y  +362.388, Z    +0.000, E1   +57.628, E3 +246967.957}
SPL {X  -163.867, Y  +354.258, Z    +0.000, E1   +57.359, E3 +246980.174}
SPL {X  -162.678, Y  +347.264, Z    +0.000, E1   +57.150, E3 +246990.515}
SPL {X  -161.618, Y  +342.173, Z    +0.000, E1   +56.783, E3 +246999.400}
SPL {X  -159.878, Y  +335.155, Z    +0.000, E1   +56.685, E3 +247009.204}
SPL {X  -158.009, Y  +328.771, Z    +0.000, E1   +56.325, E3 +247019.564}
SPL {X  -156.065, Y  +322.971, Z    +0.000, E1   +56.177, E3 +247027.908}
SPL {X  -154.487, Y  +318.719, Z    +0.000, E1   +55.733, E3 +247035.916}
SPL {X  -151.902, Y  +312.426, Z    +0.000, E1   +55.494, E3 +247045.391}
SPL {X  -149.742, Y  +307.668, Z    +0.000, E1   +54.896, E3 +247054.604}
SPL {X  -146.487, Y  +301.160, Z    +0.000, E1   +54.808, E3 +247063.466}
SPL {X  -133.590, Y  +280.553, Z    +0.000, E1   +59.642, E3 +247064.423}
SPL {X  -112.638, Y  +257.040, Z    +0.000, E1   +51.417, E3 +247167.806}
ENDSPLINE

SPLINE
SPL {X  -115.209, Y  +259.476, Z    +0.000, E1   +49.595, E3 +247201.077}
SPL {X  -147.344, Y  +302.806, Z    +0.000, E1   +40.158, E3 +247290.539}
SPL {X  -160.798, Y  +338.700, Z    +0.000, E1   +25.294, E3 +247290.021}
SPL {X  -163.893, Y  +354.439, Z    +0.000, E1   +16.805, E3 +247284.495}
SPL {X  -165.158, Y  +365.746, Z    +0.000, E1   +10.198, E3 +247282.438}
SPL {X  -165.639, Y  +376.620, Z    +0.000, E1    +3.186, E3 +247282.238}
SPL {X  -165.650, Y  +380.533, Z    +0.000, E1    +0.120, E3 +247281.266}
SPL {X  -165.650, Y  +383.454, Z    +0.000, E1    -2.667, E3 +247280.673}
SPL {X  -165.650, Y  +388.792, Z    +0.000, E1    -9.482, E3 +247279.767}
SPL {X  -165.650, Y  +393.970, Z    +0.000, E1   -17.146, E3 +247278.923}
SPL {X  -165.650, Y  +401.614, Z    +0.000, E1   -27.619, E3 +247279.579}
SPL {X  -165.650, Y  +418.105, Z    +0.000, E1   -49.413, E3 +247274.986}
SPL {X  -165.650, Y  +465.736, Z    +0.000, E1   -65.678, E3 +247288.729}
SPL {X  -165.650, Y  +519.483, Z    +0.000, E1   -68.357, E3 +247314.914}
SPL {X  -165.650, Y  +548.869, Z    +0.000, E1   -62.199, E3 +247370.606}
ENDSPLINE

SPLINE
SPL {X  -165.650, Y  +534.780, Z    +0.000, E1   -57.803, E3 +247384.256}
ENDSPLINE

SPLINE
SPL {X  -165.650, Y  +545.905, Z    +0.000, E1   -57.853, E3 +247398.195}
SPL {X  -165.650, Y  +553.630, Z    +0.000, E1   -57.616, E3 +247409.645}
SPL {X  -165.650, Y  +563.473, Z    +0.000, E1   -57.690, E3 +247422.009}
SPL {X  -165.650, Y  +573.011, Z    +0.000, E1   -57.610, E3 +247434.800}
SPL {X  -165.650, Y  +581.530, Z    +0.000, E1   -57.678, E3 +247445.398}
SPL {X  -165.650, Y  +589.475, Z    +0.000, E1   -57.572, E3 +247456.385}
SPL {X  -165.650, Y  +599.695, Z    +0.000, E1   -57.964, E3 +247467.001}
SPL {X  -165.650, Y  +606.915, Z    +0.000, E1   -57.651, E3 +247478.358}
SPL {X  -165.650, Y  +614.927, Z    +0.000, E1   -57.517, E3 +247489.628}
SPL {X  -165.650, Y  +624.337, Z    +0.000, E1   -57.671, E3 +247500.853}
SPL {X  -165.650, Y  +634.236, Z    +0.000, E1   -57.671, E3 +247513.704}
SPL {X  -165.650, Y  +647.519, Z    +0.000, E1   -57.817, E3 +247530.031}
SPL {X  -165.650, Y  +657.986, Z    +0.000, E1   -57.646, E3 +247544.467}
SPL {X  -165.650, Y  +667.585, Z    +0.000, E1   -57.803, E3 +247555.863}
SPL {X  -165.634, Y  +677.794, Z    +0.000, E1   -57.650, E3 +247570.165}
SPL {X  -165.167, Y  +688.139, Z    +0.000, E1   -57.463, E3 +247584.744}
SPL {X  -164.009, Y  +698.761, Z    +0.000, E1   -57.613, E3 +247597.517}
SPL {X  -162.382, Y  +708.242, Z    +0.000, E1   -57.205, E3 +247612.443}
SPL {X  -160.577, Y  +716.182, Z    +0.000, E1   -56.676, E3 +247625.837}
SPL {X  -158.520, Y  +723.576, Z    +0.000, E1   -56.758, E3 +247634.882}
SPL {X  -156.858, Y  +728.749, Z    +0.000, E1   -56.333, E3 +247644.024}
SPL {X  -155.155, Y  +733.525, Z    +0.000, E1   -55.869, E3 +247652.801}
SPL {X  -153.442, Y  +737.914, Z    +0.000, E1   -55.562, E3 +247660.205}
SPL {X  -150.574, Y  +744.547, Z    +0.000, E1   -55.310, E3 +247670.188}
SPL {X  -147.713, Y  +750.471, Z    +0.000, E1   -54.514, E3 +247681.851}
SPL {X  -139.786, Y  +764.381, Z    +0.000, E1   -57.209, E3 +247686.039}
SPL {X  -110.324, Y  +799.066, Z    +0.000, E1   -54.396, E3 +247754.613}
SPL {X  -100.308, Y  +807.326, Z    +0.000, E1   -52.880, E3 +247799.180}
ENDSPLINE

SPLINE
SPL {X  -108.196, Y  +800.934, Z    +0.000, E1   -52.068, E3 +247891.507}
SPL {X  -144.673, Y  +756.182, Z    +0.000, E1   -41.752, E3 +247909.586}
SPL {X  -160.601, Y  +716.087, Z    +0.000, E1   -25.730, E3 +247909.213}
SPL {X  -164.850, Y  +691.761, Z    +0.000, E1   -12.424, E3 +247906.481}
SPL {X  -165.596, Y  +679.730, Z    +0.000, E1    -4.777, E3 +247905.354}
SPL {X  -165.650, Y  +674.376, Z    +0.000, E1    -0.866, E3 +247905.270}
SPL {X  -165.650, Y  +672.384, Z    +0.000, E1    +0.908, E3 +247904.151}
SPL {X  -165.650, Y  +669.093, Z    +0.000, E1    +4.549, E3 +247904.002}
SPL {X  -165.650, Y  +663.273, Z    +0.000, E1   +12.448, E3 +247903.239}
SPL {X  -165.650, Y  +654.885, Z    +0.000, E1   +25.204, E3 +247901.791}
SPL {X  -165.650, Y  +641.882, Z    +0.000, E1   +46.566, E3 +247894.662}
SPL {X  -165.650, Y  +630.946, Z    +0.000, E1   +55.779, E3 +247895.337}
SPL {X  -165.650, Y  +595.858, Z    +0.000, E1   +64.262, E3 +247910.218}
SPL {X  -165.650, Y  +589.368, Z    +0.000, E1   +58.232, E3 +247930.959}
SPL {X  -165.650, Y  +491.251, Z    +0.000, E1   +65.373, E3 +247987.386}
ENDSPLINE

SPLINE
SPL {X  -165.650, Y  +516.236, Z    +0.000, E1   +58.457, E3 +248008.066}
ENDSPLINE

SPLINE
SPL {X  -165.650, Y  +506.715, Z    +0.000, E1   +58.090, E3 +248022.519}
SPL {X  -165.650, Y  +496.085, Z    +0.000, E1   +57.984, E3 +248036.767}
SPL {X  -165.650, Y  +485.167, Z    +0.000, E1   +58.003, E3 +248050.599}
ENDSPLINE

SPLINE
SPL {X  -165.650, Y  +505.180, Z    +0.000, E1   +52.333, E3 +248057.351}
SPL {X  -165.650, Y  +506.534, Z    +0.000, E1   +50.148, E3 +248068.810}
ENDSPLINE

SPLINE
SPL {X  -165.650, Y  +495.166, Z    +0.000, E1   +51.070, E3 +248082.239}
SPL {X  -165.650, Y  +485.807, Z    +0.000, E1   +51.973, E3 +248091.971}
SPL {X  -165.650, Y  +475.672, Z    +0.000, E1   +52.573, E3 +248104.425}
SPL {X  -165.650, Y  +459.814, Z    +0.000, E1   +53.888, E3 +248120.614}
SPL {X  -165.650, Y  +448.876, Z    +0.000, E1   +54.452, E3 +248133.109}
SPL {X  -165.650, Y  +440.843, Z    +0.000, E1   +55.023, E3 +248141.174}
SPL {X  -165.650, Y  +431.771, Z    +0.000, E1   +55.549, E3 +248150.691}
SPL {X  -165.650, Y  +420.799, Z    +0.000, E1   +56.452, E3 +248160.077}
SPL {X  -165.650, Y  +409.731, Z    +0.000, E1   +57.273, E3 +248169.565}
SPL {X  -165.650, Y  +399.687, Z    +0.000, E1   +57.433, E3 +248181.750}
SPL {X  -165.650, Y  +388.492, Z    +0.000, E1   +57.709, E3 +248194.463}
SPL {X  -165.650, Y  +379.894, Z    +0.000, E1   +57.709, E3 +248205.567}
SPL {X  -165.538, Y  +372.423, Z    +0.000, E1   +57.528, E3 +248216.440}
SPL {X  -164.865, Y  +362.388, Z    +0.000, E1   +57.628, E3 +248228.826}
SPL {X  -163.867, Y  +354.258, Z    +0.000, E1   +57.359, E3 +248241.043}
SPL {X  -162.678, Y  +347.264, Z    +0.000, E1   +57.150, E3 +248251.384}
SPL {X  -161.618, Y  +342.173, Z    +0.000, E1   +56.783, E3 +248260.270}
SPL {X  -159.878, Y  +335.155, Z    +0.000, E1   +56.685, E3 +248270.074}
SPL {X  -158.009, Y  +328.771, Z    +0.000, E1   +56.325, E3 +248280.433}
SPL {X  -156.065, Y  +322.971, Z    +0.000, E1   +56.177, E3 +248288.777}
SPL {X  -154.487, Y  +318.719, Z    +0.000, E1   +55.733, E3 +248296.786}
SPL {X  -151.902, Y  +312.426, Z    +0.000, E1   +55.494, E3 +248306.261}
SPL {X  -149.742, Y  +307.668, Z    +0.000, E1   +54.896, E3 +248315.473}
SPL {X  -146.487, Y  +301.160, Z    +0.000, E1   +54.808, E3 +248324.336}
SPL {X  -133.590, Y  +280.553, Z    +0.000, E1   +59.642, E3 +248325.293}
SPL {X  -112.638, Y  +257.040, Z    +0.000, E1   +51.417, E3 +248428.676}
ENDSPLINE

SPLINE
SPL {X  -115.209, Y  +259.476, Z    +0.000, E1   +49.595, E3 +248461.946}
SPL {X  -147.344, Y  +302.806, Z    +0.000, E1   +40.158, E3 +248551.409}
SPL {X  -160.798, Y  +338.700, Z    +0.000, E1   +25.294, E3 +248550.890}
SPL {X  -163.893, Y  +354.439, Z    +0.000, E1   +16.805, E3 +248545.365}
SPL {X  -165.158, Y  +365.746, Z    +0.000, E1   +10.198, E3 +248543.307}
SPL {X  -165.639, Y  +376.620, Z    +0.000, E1    +3.186, E3 +248543.107}
SPL {X  -165.650, Y  +381.477, Z    +0.000, E1    -0.622, E3 +248541.918}
SPL {X  -165.650, Y  +384.861, Z    +0.000, E1    -4.465, E3 +248541.320}
SPL {X  -165.650, Y  +388.792, Z    +0.000, E1    -9.482, E3 +248540.637}
SPL {X  -165.650, Y  +393.970, Z    +0.000, E1   -17.146, E3 +248539.793}
SPL {X  -165.650, Y  +401.614, Z    +0.000, E1   -27.619, E3 +248540.448}
SPL {X  -165.650, Y  +418.105, Z    +0.000, E1   -49.413, E3 +248535.856}
SPL {X  -165.650, Y  +465.736, Z    +0.000, E1   -65.678, E3 +248549.599}
SPL {X  -165.650, Y  +519.483, Z    +0.000, E1   -68.357, E3 +248575.783}
SPL {X  -165.650, Y  +548.869, Z    +0.000, E1   -62.199, E3 +248631.476}
ENDSPLINE

SPLINE
SPL {X  -165.650, Y  +534.780, Z    +0.000, E1   -57.803, E3 +248645.125}
ENDSPLINE

SPLINE
SPL {X  -165.650, Y  +545.905, Z    +0.000, E1   -57.853, E3 +248659.065}
SPL {X  -165.650, Y  +555.746, Z    +0.000, E1   -57.571, E3 +248673.702}
SPL {X  -165.650, Y  +566.557, Z    +0.000, E1   -57.834, E3 +248685.830}
SPL {X  -165.650, Y  +573.011, Z    +0.000, E1   -57.610, E3 +248695.670}
SPL {X  -165.650, Y  +581.530, Z    +0.000, E1   -57.678, E3 +248706.268}
SPL {X  -165.650, Y  +589.475, Z    +0.000, E1   -57.572, E3 +248717.255}
SPL {X  -165.650, Y  +599.695, Z    +0.000, E1   -57.964, E3 +248727.871}
SPL {X  -165.650, Y  +606.915, Z    +0.000, E1   -57.651, E3 +248739.227}
SPL {X  -165.650, Y  +614.927, Z    +0.000, E1   -57.517, E3 +248750.497}
SPL {X  -165.650, Y  +624.337, Z    +0.000, E1   -57.671, E3 +248761.723}
SPL {X  -165.650, Y  +634.236, Z    +0.000, E1   -57.671, E3 +248774.573}
SPL {X  -165.650, Y  +647.519, Z    +0.000, E1   -57.817, E3 +248790.901}
SPL {X  -165.650, Y  +657.986, Z    +0.000, E1   -57.646, E3 +248805.336}
SPL {X  -165.650, Y  +667.585, Z    +0.000, E1   -57.803, E3 +248816.732}
SPL {X  -165.634, Y  +677.794, Z    +0.000, E1   -57.650, E3 +248831.034}
SPL {X  -165.167, Y  +688.139, Z    +0.000, E1   -57.463, E3 +248845.614}
SPL {X  -164.323, Y  +696.426, Z    +0.000, E1   -57.565, E3 +248855.600}
SPL {X  -163.313, Y  +703.224, Z    +0.000, E1   -57.403, E3 +248865.494}
SPL {X  -161.906, Y  +710.520, Z    +0.000, E1   -57.149, E3 +248876.446}
SPL {X  -160.577, Y  +716.182, Z    +0.000, E1   -56.676, E3 +248886.706}
SPL {X  -158.520, Y  +723.576, Z    +0.000, E1   -56.758, E3 +248895.751}
SPL {X  -156.858, Y  +728.749, Z    +0.000, E1   -56.333, E3 +248904.894}
SPL {X  -155.155, Y  +733.525, Z    +0.000, E1   -55.869, E3 +248913.670}
SPL {X  -152.530, Y  +740.111, Z    +0.000, E1   -55.545, E3 +248924.147}
SPL {X  -149.838, Y  +746.130, Z    +0.000, E1   -55.135, E3 +248933.867}
SPL {X  -147.713, Y  +750.471, Z    +0.000, E1   -54.514, E3 +248942.720}
SPL {X  -139.786, Y  +764.381, Z    +0.000, E1   -57.209, E3 +248946.908}
SPL {X  -110.324, Y  +799.066, Z    +0.000, E1   -54.396, E3 +249015.482}
SPL {X  -100.308, Y  +807.326, Z    +0.000, E1   -52.880, E3 +249060.050}
ENDSPLINE

SPLINE
SPL {X  -108.196, Y  +800.934, Z    +0.000, E1   -52.068, E3 +249152.376}
SPL {X  -144.673, Y  +756.182, Z    +0.000, E1   -41.752, E3 +249170.455}
SPL {X  -158.838, Y  +722.515, Z    +0.000, E1   -28.697, E3 +249169.939}
SPL {X  -163.562, Y  +701.720, Z    +0.000, E1   -18.114, E3 +249167.153}
SPL {X  -165.078, Y  +689.251, Z    +0.000, E1   -10.876, E3 +249168.705}
SPL {X  -165.596, Y  +679.730, Z    +0.000, E1    -4.777, E3 +249166.224}
SPL {X  -165.650, Y  +674.376, Z    +0.000, E1    -0.866, E3 +249166.139}
SPL {X  -165.650, Y  +672.384, Z    +0.000, E1    +0.908, E3 +249165.020}
SPL {X  -165.650, Y  +669.093, Z    +0.000, E1    +4.549, E3 +249164.872}
SPL {X  -165.650, Y  +663.273, Z    +0.000, E1   +12.448, E3 +249164.109}
SPL {X  -165.650, Y  +654.885, Z    +0.000, E1   +25.204, E3 +249162.661}
SPL {X  -165.650, Y  +641.882, Z    +0.000, E1   +46.566, E3 +249155.532}
SPL {X  -165.650, Y  +630.946, Z    +0.000, E1   +55.779, E3 +249156.206}
SPL {X  -165.650, Y  +595.858, Z    +0.000, E1   +64.262, E3 +249171.087}
SPL {X  -165.650, Y  +589.368, Z    +0.000, E1   +58.232, E3 +249191.829}
SPL {X  -165.650, Y  +491.251, Z    +0.000, E1   +65.373, E3 +249248.255}
ENDSPLINE

SPLINE
SPL {X  -165.650, Y  +516.236, Z    +0.000, E1   +58.457, E3 +249268.936}
ENDSPLINE

SPLINE
SPL {X  -165.650, Y  +506.715, Z    +0.000, E1   +58.090, E3 +249283.389}
SPL {X  -165.650, Y  +496.085, Z    +0.000, E1   +57.984, E3 +249297.636}
SPL {X  -165.650, Y  +485.167, Z    +0.000, E1   +58.003, E3 +249311.468}
ENDSPLINE

SPLINE
SPL {X  -165.650, Y  +509.193, Z    +0.000, E1   +50.604, E3 +249322.435}
ENDSPLINE

